C07281=1128.691,-66.097,-47.066,178.905,6.216,149.446
C07282=1128.696,-66.348,-47.056,178.902,6.216,149.447
C07283=1128.701,-66.597,-47.046,178.900,6.215,149.447
C07284=1128.707,-66.847,-47.035,178.898,6.215,149.448
C07285=1128.712,-67.097,-47.025,178.896,6.214,149.448
C07286=1128.717,-67.347,-47.015,178.893,6.213,149.449
C07287=1128.722,-67.596,-47.005,178.892,6.213,149.449
C07288=1128.727,-67.846,-46.994,178.890,6.212,149.450
C07289=1128.733,-68.096,-46.984,178.887,6.212,149.451
C07290=1128.739,-68.345,-46.974,178.885,6.211,149.451
C07291=1128.744,-68.595,-46.963,178.882,6.210,149.452
C07292=1128.749,-68.846,-46.954,178.880,6.210,149.452
C07293=1128.754,-69.095,-46.944,178.879,6.210,149.452
C07294=1128.760,-69.344,-46.934,178.877,6.209,149.453
C07295=1128.765,-69.595,-46.923,178.874,6.209,149.454
C07296=1128.770,-69.844,-46.913,178.872,6.208,149.454
C07297=1128.776,-70.094,-46.903,178.869,6.207,149.455
C07298=1128.781,-70.343,-46.893,178.867,6.206,149.455
C07299=1128.786,-70.593,-46.883,178.866,6.206,149.456
C07300=1128.792,-70.843,-46.873,178.863,6.206,149.456
C07301=1128.797,-71.093,-46.863,178.861,6.205,149.457
C07302=1128.802,-71.342,-46.854,178.859,6.204,149.457
C07303=1128.807,-71.592,-46.843,178.856,6.204,149.458
C07304=1128.813,-71.842,-46.833,178.855,6.204,149.458
C07305=1128.818,-72.091,-46.823,178.853,6.203,149.459
C07306=1128.824,-72.341,-46.814,178.850,6.202,149.459
C07307=1128.829,-72.591,-46.803,178.848,6.201,149.460
C07308=1128.834,-72.841,-46.793,178.846,6.201,149.460
C07309=1128.840,-73.091,-46.783,178.844,6.201,149.461
C07310=1128.845,-73.340,-46.773,178.842,6.200,149.461
C07311=1128.851,-73.590,-46.764,178.840,6.200,149.462
C07312=1128.856,-73.840,-46.753,178.837,6.199,149.462
C07313=1128.860,-74.089,-46.743,178.835,6.198,149.463
C07314=1128.866,-74.339,-46.733,178.834,6.198,149.463
C07315=1128.872,-74.589,-46.724,178.831,6.197,149.464
C07316=1128.877,-74.839,-46.713,178.829,6.197,149.464
C07317=1128.882,-75.089,-46.703,178.827,6.196,149.465
C07318=1128.887,-75.338,-46.693,178.824,6.195,149.465
C07319=1128.893,-75.588,-46.684,178.823,6.196,149.466
C07320=1128.898,-75.838,-46.674,178.821,6.195,149.466
C07321=1128.904,-76.087,-46.664,178.818,6.194,149.467
C07322=1128.909,-76.338,-46.654,178.816,6.193,149.467
C07323=1128.914,-76.587,-46.644,178.814,6.192,149.468
C07324=1128.920,-76.858,-46.633,178.812,6.193,149.469
C07325=1128.926,-77.130,-46.623,178.810,6.192,149.469
C07326=1128.931,-77.401,-46.612,178.808,6.191,149.470
C07327=1128.937,-77.674,-46.601,178.805,6.191,149.470
C07328=1128.943,-77.923,-46.591,178.803,6.190,149.471
C07329=1128.948,-78.173,-46.582,178.800,6.190,149.471
C07330=1128.954,-78.422,-46.572,178.798,6.189,149.472
C07331=1128.959,-78.672,-46.562,178.797,6.189,149.472
C07332=1128.965,-78.922,-46.553,178.794,6.188,149.473
C07333=1128.970,-79.171,-46.543,178.792,6.187,149.473
C07334=1128.975,-79.422,-46.533,178.790,6.187,149.474
C07335=1128.980,-79.672,-46.523,178.788,6.187,149.474
C07336=1128.985,-79.921,-46.514,178.786,6.186,149.475
C07337=1128.991,-80.171,-46.504,178.784,6.185,149.475
C07338=1128.997,-80.420,-46.494,178.781,6.185,149.476
C07339=1129.002,-80.670,-46.485,178.779,6.184,149.476
C07340=1129.007,-80.920,-46.475,178.778,6.184,149.477
C07341=1129.012,-81.169,-46.465,178.775,6.183,149.477
C07342=1129.018,-81.420,-46.455,178.773,6.183,149.478
C07343=1129.022,-81.669,-46.446,178.771,6.182,149.478
C07344=1129.028,-81.919,-46.436,178.769,6.182,149.479
C07345=1129.033,-82.169,-46.427,178.767,6.181,149.479
C07346=1129.039,-82.419,-46.417,178.765,6.181,149.480
C07347=1129.044,-82.668,-46.408,178.762,6.180,149.480
C07348=1129.050,-82.918,-46.398,178.761,6.180,149.481
C07349=1129.055,-83.168,-46.388,178.759,6.179,149.481
C07350=1129.061,-83.418,-46.379,178.756,6.178,149.482
C07351=1129.066,-83.667,-46.369,178.754,6.178,149.482
C07352=1129.071,-83.918,-46.359,178.753,6.178,149.483
C07353=1129.076,-84.167,-46.349,178.750,6.177,149.483
C07354=1129.082,-84.417,-46.340,178.748,6.176,149.484
C07355=1129.087,-84.667,-46.330,178.747,6.176,149.484
C07356=1129.092,-84.916,-46.321,178.744,6.176,149.485
C07357=1129.097,-85.166,-46.312,178.742,6.175,149.485
C07358=1129.103,-85.416,-46.302,178.740,6.174,149.486
C07359=1129.108,-85.665,-46.293,178.738,6.174,149.486
C07360=1129.114,-85.915,-46.283,178.736,6.174,149.487
C07361=1129.119,-86.165,-46.274,178.734,6.173,149.487
C07362=1129.125,-86.415,-46.264,178.731,6.172,149.488
C07363=1129.130,-86.664,-46.255,178.730,6.172,149.488
C07364=1129.135,-86.914,-46.245,178.728,6.171,149.489
C07365=1129.141,-87.164,-46.236,178.725,6.171,149.489
C07366=1129.146,-87.414,-46.227,178.723,6.170,149.490
C07367=1129.151,-87.663,-46.217,178.722,6.170,149.490
C07368=1129.156,-87.913,-46.208,178.719,6.170,149.491
C07369=1129.162,-88.163,-46.198,178.717,6.169,149.492
C07370=1129.167,-88.412,-46.189,178.715,6.169,149.492
C07371=1129.173,-88.663,-46.179,178.713,6.168,149.492
C07372=1129.178,-88.912,-46.170,178.711,6.167,149.493
C07373=1129.183,-89.162,-46.161,178.709,6.167,149.493
C07374=1129.189,-89.412,-46.151,178.707,6.167,149.494
C07375=1129.194,-89.661,-46.142,178.705,6.166,149.494
C07376=1129.199,-89.911,-46.133,178.703,6.165,149.495
C07377=1129.205,-90.161,-46.123,178.701,6.165,149.495
C07378=1129.210,-90.410,-46.114,178.699,6.165,149.496
C07379=1129.216,-90.661,-46.104,178.697,6.164,149.496
C07380=1129.221,-90.910,-46.095,178.695,6.164,149.497
C07381=1129.226,-91.160,-46.086,178.693,6.163,149.497
C07382=1129.232,-91.410,-46.076,178.690,6.163,149.498
C07383=1129.237,-91.660,-46.067,178.688,6.162,149.499
C07384=1129.242,-91.909,-46.058,178.686,6.162,149.499
C07385=1129.248,-92.159,-46.048,178.684,6.161,149.499
C07386=1129.253,-92.409,-46.039,178.682,6.161,149.500
C07387=1129.258,-92.659,-46.030,178.680,6.161,149.500
C07388=1129.264,-92.909,-46.021,178.678,6.160,149.501
C07389=1129.269,-93.158,-46.011,178.676,6.159,149.501
C07390=1129.274,-93.408,-46.002,178.674,6.159,149.502
C07391=1129.280,-93.658,-45.993,178.672,6.158,149.502
C07392=1129.285,-93.908,-45.984,178.670,6.158,149.503
C07393=1129.290,-94.157,-45.974,178.668,6.158,149.503
C07394=1129.296,-94.407,-45.965,178.666,6.157,149.504
C07395=1129.301,-94.657,-45.956,178.664,6.156,149.504
C07396=1129.306,-94.907,-45.947,178.662,6.155,149.505
C07397=1129.311,-95.157,-45.938,178.660,6.155,149.505
C07398=1129.317,-95.406,-45.928,178.658,6.155,149.506
C07399=1129.322,-95.656,-45.919,178.656,6.154,149.506
C07400=1129.328,-95.905,-45.911,178.654,6.154,149.507
C07401=1129.334,-96.156,-45.901,178.652,6.153,149.507
C07402=1129.339,-96.405,-45.892,178.649,6.153,149.508
C07403=1129.344,-96.655,-45.883,178.648,6.153,149.508
C07404=1129.349,-96.905,-45.874,178.646,6.152,149.509
C07405=1129.355,-97.155,-45.864,178.643,6.151,149.509
C07406=1129.360,-97.405,-45.855,178.642,6.151,149.510
C07407=1129.365,-97.654,-45.846,178.640,6.151,149.510
C07408=1129.370,-97.904,-45.837,178.637,6.150,149.511
C07409=1129.375,-98.154,-45.829,178.636,6.150,149.511
C07410=1129.382,-98.404,-45.819,178.634,6.149,149.512
C07411=1129.387,-98.653,-45.811,178.631,6.149,149.512
C07412=1129.392,-98.903,-45.802,178.630,6.149,149.513
C07413=1129.397,-99.153,-45.793,178.628,6.148,149.513
C07414=1129.403,-99.403,-45.783,178.625,6.147,149.514
C07415=1129.408,-99.653,-45.774,178.624,6.147,149.514
C07416=1129.413,-99.902,-45.765,178.622,6.146,149.515
C07417=1129.419,-100.152,-45.756,178.619,6.146,149.515
C07418=1129.424,-100.401,-45.747,178.618,6.146,149.516
C07419=1129.430,-100.652,-45.738,178.616,6.145,149.516
C07420=1129.435,-100.901,-45.729,178.614,6.145,149.517
C07421=1129.441,-101.151,-45.720,178.612,6.144,149.517
C07422=1129.446,-101.401,-45.711,178.610,6.143,149.518
C07423=1129.451,-101.651,-45.702,178.608,6.144,149.518
C07424=1129.457,-101.900,-45.694,178.606,6.143,149.519
C07425=1129.462,-102.150,-45.685,178.604,6.142,149.519
C07426=1129.468,-102.400,-45.675,178.602,6.142,149.520
C07427=1129.473,-102.650,-45.666,178.600,6.141,149.520
C07428=1129.479,-102.923,-45.657,178.598,6.141,149.521
C07429=1129.484,-103.195,-45.647,178.595,6.140,149.521
C07430=1129.490,-103.467,-45.637,178.593,6.140,149.522
C07431=1129.496,-103.739,-45.628,178.591,6.140,149.522
C07432=1129.502,-103.989,-45.619,178.589,6.139,149.523
C07433=1129.507,-104.239,-45.610,178.587,6.139,149.523
C07434=1129.512,-104.488,-45.601,178.585,6.138,149.524
C07435=1129.517,-104.738,-45.592,178.583,6.137,149.524
C07436=1129.523,-104.987,-45.584,178.581,6.137,149.525
C07437=1129.529,-105.238,-45.574,178.579,6.137,149.525
C07438=1129.534,-105.488,-45.566,178.577,6.136,149.526
C07439=1129.539,-105.738,-45.557,178.575,6.136,149.526
C07440=1129.545,-105.988,-45.548,178.573,6.135,149.527
C07441=1129.550,-106.237,-45.540,178.572,6.135,149.527
C07442=1129.555,-106.487,-45.531,178.569,6.135,149.528
C07443=1129.561,-106.737,-45.522,178.567,6.134,149.528
C07444=1129.566,-106.986,-45.513,178.566,6.134,149.529
C07445=1129.571,-107.236,-45.504,178.563,6.133,149.529
C07446=1129.577,-107.485,-45.496,178.561,6.132,149.530
C07447=1129.582,-107.736,-45.488,178.560,6.132,149.530
C07448=1129.587,-107.986,-45.479,178.557,6.132,149.531
C07449=1129.593,-108.236,-45.470,178.556,6.132,149.531
C07450=1129.598,-108.485,-45.461,178.554,6.131,149.532
C07451=1129.603,-108.735,-45.452,178.551,6.130,149.532
C07452=1129.609,-108.984,-45.443,178.550,6.130,149.533
C07453=1129.614,-109.235,-45.435,178.548,6.130,149.533
C07454=1129.620,-109.484,-45.427,178.546,6.130,149.533
C07455=1129.625,-109.734,-45.418,178.544,6.128,149.534
C07456=1129.630,-109.984,-45.409,178.542,6.128,149.534
C07457=1129.635,-110.234,-45.400,178.540,6.128,149.535
C07458=1129.641,-110.483,-45.392,178.538,6.127,149.535
C07459=1129.647,-110.733,-45.383,178.537,6.127,149.536
C07460=1129.652,-110.983,-45.374,178.535,6.126,149.536
C07461=1129.658,-111.232,-45.366,178.532,6.126,149.537
C07462=1129.663,-111.483,-45.358,178.531,6.126,149.537
C07463=1129.668,-111.733,-45.349,178.529,6.125,149.538
C07464=1129.673,-111.982,-45.340,178.527,6.125,149.538
C07465=1129.679,-112.232,-45.331,178.525,6.124,149.539
C07466=1129.685,-112.482,-45.323,178.523,6.123,149.539
C07467=1129.690,-112.732,-45.314,178.521,6.123,149.540
C07468=1129.696,-112.981,-45.306,178.519,6.123,149.540
C07469=1129.701,-113.231,-45.297,178.517,6.123,149.541
C07470=1129.706,-113.481,-45.289,178.515,6.122,149.541
C07471=1129.711,-113.731,-45.280,178.513,6.122,149.542
C07472=1129.717,-113.980,-45.271,178.511,6.121,149.542
C07473=1129.723,-114.231,-45.263,178.509,6.121,149.543
C07474=1129.728,-114.481,-45.254,178.507,6.121,149.543
C07475=1129.734,-114.730,-45.246,178.505,6.120,149.543
C07476=1129.738,-114.980,-45.238,178.504,6.120,149.544
C07477=1129.743,-115.230,-45.229,178.502,6.119,149.544
C07478=1129.749,-115.479,-45.221,178.500,6.118,149.545
C07479=1129.755,-115.729,-45.212,178.498,6.118,149.545
C07480=1129.760,-115.979,-45.204,178.496,6.117,149.546
C07481=1129.766,-116.228,-45.195,178.494,6.117,149.546
C07482=1129.771,-116.479,-45.187,178.492,6.117,149.547
C07483=1129.776,-116.729,-45.178,178.490,6.117,149.547
C07484=1129.782,-116.978,-45.169,178.488,6.116,149.548
C07485=1129.787,-117.228,-45.161,178.486,6.115,149.548
C07486=1129.792,-117.477,-45.153,178.484,6.115,149.549
C07487=1129.798,-117.728,-45.145,178.482,6.115,149.549
C07488=1129.803,-117.978,-45.136,178.481,6.115,149.550
C07489=1129.809,-118.227,-45.128,178.478,6.114,149.550
C07490=1129.814,-118.477,-45.119,178.477,6.114,149.551
C07491=1129.820,-118.727,-45.111,178.475,6.113,149.551
C07492=1129.826,-118.977,-45.103,178.474,6.113,149.551
C07493=1129.830,-119.226,-45.094,178.471,6.112,149.552
C07494=1129.836,-119.475,-45.086,178.469,6.111,149.552
C07495=1129.841,-119.726,-45.078,178.468,6.111,149.553
C07496=1129.846,-119.976,-45.069,178.465,6.111,149.553
C07497=1129.853,-120.226,-45.061,178.464,6.111,149.554
C07498=1129.857,-120.475,-45.053,178.462,6.110,149.554
C07499=1129.862,-120.726,-45.045,178.460,6.110,149.555
C07500=1129.868,-120.975,-45.036,178.458,6.109,149.555
C07501=1129.874,-121.225,-45.028,178.456,6.109,149.556
C07502=1129.879,-121.474,-45.019,178.454,6.109,149.556
C07503=1129.884,-121.725,-45.012,178.453,6.108,149.556
C07504=1129.889,-121.974,-45.003,178.451,6.107,149.557
C07505=1129.895,-122.224,-44.995,178.448,6.107,149.557
C07506=1129.901,-122.474,-44.986,178.447,6.107,149.558
C07507=1129.906,-122.723,-44.979,178.445,6.106,149.558
C07508=1129.911,-122.973,-44.970,178.443,6.106,149.559
C07509=1129.917,-123.223,-44.962,178.441,6.105,149.559
C07510=1129.922,-123.473,-44.953,178.439,6.105,149.560
C07511=1129.928,-123.723,-44.945,178.437,6.105,149.560
C07512=1129.933,-123.972,-44.937,178.436,6.104,149.561
C07513=1129.938,-124.223,-44.929,178.434,6.104,149.561
C07514=1129.944,-124.472,-44.921,178.432,6.104,149.562
C07515=1129.949,-124.722,-44.913,178.430,6.103,149.562
C07516=1129.955,-124.972,-44.905,178.428,6.103,149.563
C07517=1129.960,-125.222,-44.896,178.426,6.102,149.563
C07518=1129.966,-125.471,-44.888,178.425,6.102,149.564
C07519=1129.971,-125.721,-44.880,178.422,6.102,149.564
C07520=1129.976,-125.971,-44.872,178.420,6.101,149.565
C07521=1129.982,-126.221,-44.864,178.419,6.100,149.565
C07522=1129.986,-126.471,-44.856,178.417,6.100,149.565
C07523=1129.993,-126.720,-44.848,178.415,6.100,149.566
C07524=1129.998,-126.970,-44.839,178.413,6.099,149.566
C07525=1130.004,-127.220,-44.831,178.411,6.099,149.567
C07526=1130.009,-127.470,-44.824,178.409,6.098,149.567
C07527=1130.014,-127.719,-44.815,178.408,6.098,149.568
C07528=1130.020,-127.970,-44.807,178.405,6.098,149.568
C07529=1130.025,-128.219,-44.800,178.404,6.097,149.568
C07530=1130.030,-128.469,-44.791,178.402,6.097,149.569
C07531=1130.036,-128.719,-44.783,178.401,6.097,149.569
C07532=1129.615,-128.730,-44.827,178.397,6.100,149.571
C07533=1129.610,-128.481,-44.836,178.399,6.101,149.571
C07534=1129.604,-128.230,-44.844,178.401,6.101,149.570
C07535=1129.599,-127.981,-44.851,178.403,6.101,149.570
C07536=1129.594,-127.731,-44.860,178.404,6.101,149.569
C07537=1129.587,-127.481,-44.868,178.407,6.102,149.569
C07538=1129.583,-127.231,-44.875,178.408,6.102,149.569
C07539=1129.577,-126.982,-44.884,178.410,6.103,149.568
C07540=1129.571,-126.732,-44.892,178.411,6.103,149.568
C07541=1129.567,-126.482,-44.900,178.414,6.104,149.567
C07542=1129.561,-126.232,-44.908,178.416,6.105,149.567
C07543=1129.556,-125.982,-44.916,178.417,6.104,149.566
C07544=1129.550,-125.733,-44.925,178.420,6.105,149.566
C07545=1129.545,-125.483,-44.932,178.421,6.105,149.565
C07546=1129.539,-125.233,-44.941,178.423,6.106,149.565
C07547=1129.534,-124.983,-44.949,178.425,6.106,149.564
C07548=1129.528,-124.733,-44.956,178.427,6.107,149.564
C07549=1129.523,-124.484,-44.965,178.428,6.107,149.563
C07550=1129.517,-124.234,-44.973,178.431,6.108,149.563
C07551=1129.512,-123.984,-44.982,178.432,6.108,149.562
C07552=1129.507,-123.734,-44.990,178.434,6.108,149.562
C07553=1129.502,-123.485,-44.998,178.436,6.108,149.561
C07554=1129.496,-123.234,-45.006,178.438,6.109,149.561
C07555=1129.490,-122.985,-45.015,178.439,6.109,149.561
C07556=1129.486,-122.735,-45.022,178.441,6.110,149.560
C07557=1129.479,-122.485,-45.030,178.443,6.110,149.560
C07558=1129.474,-122.235,-45.039,178.445,6.111,149.559
C07559=1129.469,-121.985,-45.047,178.447,6.112,149.559
C07560=1129.463,-121.736,-45.056,178.449,6.112,149.558
C07561=1129.458,-121.485,-45.063,178.451,6.112,149.558
C07562=1129.453,-121.236,-45.072,178.453,6.112,149.557
C07563=1129.447,-120.986,-45.081,178.455,6.113,149.557
C07564=1129.442,-120.736,-45.089,178.456,6.113,149.557
C07565=1129.437,-120.487,-45.097,178.458,6.114,149.556
C07566=1129.431,-120.237,-45.105,178.460,6.114,149.556
C07567=1129.426,-119.988,-45.114,178.462,6.115,149.555
C07568=1129.420,-119.737,-45.122,178.464,6.115,149.555
C07569=1129.415,-119.487,-45.131,178.466,6.115,149.554
C07570=1129.409,-119.237,-45.139,178.468,6.116,149.554
C07571=1129.405,-118.988,-45.147,178.470,6.116,149.553
C07572=1129.398,-118.738,-45.155,178.472,6.117,149.553
C07573=1129.393,-118.488,-45.164,178.474,6.117,149.552
C07574=1129.388,-118.238,-45.173,178.476,6.118,149.552
C07575=1129.382,-117.989,-45.180,178.477,6.118,149.551
C07576=1129.377,-117.739,-45.189,178.479,6.119,149.551
C07577=1129.372,-117.489,-45.197,178.481,6.119,149.550
C07578=1129.366,-117.240,-45.205,178.483,6.119,149.550
C07579=1129.361,-116.990,-45.214,178.485,6.120,149.549
C07580=1129.356,-116.739,-45.222,178.487,6.120,149.549
C07581=1129.350,-116.490,-45.231,178.489,6.121,149.548
C07582=1129.345,-116.240,-45.239,178.490,6.121,149.548
C07583=1129.339,-115.990,-45.248,178.493,6.121,149.548
C07584=1129.334,-115.741,-45.257,178.495,6.122,149.547
C07585=1129.328,-115.490,-45.265,178.496,6.122,149.547
C07586=1129.323,-115.241,-45.273,178.499,6.123,149.546
C07587=1129.318,-114.991,-45.282,178.500,6.123,149.546
C07588=1129.312,-114.741,-45.290,178.502,6.124,149.545
C07589=1129.307,-114.492,-45.298,178.504,6.124,149.545
C07590=1129.301,-114.242,-45.307,178.506,6.125,149.544
C07591=1129.296,-113.991,-45.315,178.508,6.125,149.544
C07592=1129.291,-113.742,-45.324,178.510,6.125,149.543
C07593=1129.285,-113.492,-45.333,178.512,6.126,149.543
C07594=1129.280,-113.243,-45.342,178.513,6.126,149.542
C07595=1129.274,-112.992,-45.350,178.516,6.127,149.542
C07596=1129.269,-112.743,-45.358,178.517,6.127,149.541
C07597=1129.264,-112.493,-45.367,178.519,6.127,149.541
C07598=1129.258,-112.243,-45.376,178.522,6.128,149.540
C07599=1129.252,-111.994,-45.384,178.523,6.128,149.540
C07600=1129.247,-111.744,-45.393,178.525,6.129,149.539
C07601=1129.242,-111.494,-45.402,178.527,6.129,149.539
C07602=1129.236,-111.243,-45.410,178.529,6.130,149.538
C07603=1129.231,-110.995,-45.418,178.531,6.130,149.538
C07604=1129.226,-110.745,-45.427,178.533,6.130,149.538
C07605=1129.221,-110.495,-45.436,178.535,6.131,149.537
C07606=1129.215,-110.245,-45.444,178.537,6.131,149.537
C07607=1129.210,-109.995,-45.452,178.539,6.132,149.536
C07608=1129.205,-109.745,-45.461,178.541,6.132,149.536
C07609=1129.200,-109.495,-45.470,178.543,6.132,149.535
C07610=1129.194,-109.246,-45.479,178.545,6.133,149.535
C07611=1129.189,-108.997,-45.488,178.546,6.134,149.534
C07612=1129.183,-108.746,-45.496,178.548,6.134,149.534
C07613=1129.178,-108.496,-45.505,178.550,6.135,149.533
C07614=1129.171,-108.247,-45.514,178.552,6.135,149.533
C07615=1129.166,-107.997,-45.523,178.554,6.136,149.532
C07616=1129.161,-107.747,-45.532,178.556,6.136,149.532
C07617=1129.156,-107.497,-45.541,178.558,6.136,149.531
C07618=1129.150,-107.247,-45.548,178.560,6.137,149.531
C07619=1129.145,-106.998,-45.557,178.562,6.137,149.530
C07620=1129.140,-106.748,-45.566,178.564,6.138,149.530
C07621=1129.134,-106.498,-45.575,178.566,6.139,149.529
C07622=1129.129,-106.248,-45.584,178.568,6.139,149.529
C07623=1129.123,-105.999,-45.593,178.570,6.139,149.528
C07624=1129.118,-105.749,-45.601,178.572,6.139,149.528
C07625=1129.113,-105.499,-45.610,178.574,6.140,149.528
C07626=1129.108,-105.249,-45.619,178.576,6.141,149.527
C07627=1129.102,-105.000,-45.627,178.578,6.141,149.527
C07628=1129.097,-104.750,-45.636,178.580,6.141,149.526
C07629=1129.092,-104.500,-45.645,178.582,6.142,149.526
C07630=1129.086,-104.250,-45.654,178.584,6.142,149.525
C07631=1129.080,-104.000,-45.663,178.586,6.143,149.525
C07632=1129.075,-103.750,-45.672,178.587,6.143,149.524
C07633=1129.069,-103.478,-45.681,178.590,6.144,149.524
C07634=1129.063,-103.206,-45.692,178.592,6.144,149.523
C07635=1129.058,-102.934,-45.701,178.594,6.145,149.522
C07636=1129.052,-102.661,-45.711,178.597,6.145,149.522
C07637=1129.047,-102.411,-45.719,178.598,6.145,149.521
C07638=1129.041,-102.161,-45.728,178.600,6.146,149.521
C07639=1129.036,-101.912,-45.737,178.603,6.147,149.520
C07640=1129.030,-101.662,-45.746,178.604,6.147,149.520
C07641=1129.025,-101.412,-45.755,178.606,6.148,149.519
C07642=1129.019,-101.162,-45.764,178.608,6.147,149.519
C07643=1129.014,-100.913,-45.773,178.610,6.148,149.519
C07644=1129.009,-100.663,-45.782,178.612,6.149,149.518
C07645=1129.004,-100.413,-45.791,178.614,6.149,149.518
C07646=1128.997,-100.163,-45.800,178.616,6.150,149.517
C07647=1128.992,-99.913,-45.809,178.618,6.150,149.517
C07648=1128.987,-99.664,-45.818,178.620,6.150,149.516
C07649=1128.982,-99.414,-45.827,178.622,6.151,149.516
C07650=1128.977,-99.165,-45.836,178.624,6.152,149.515
C07651=1128.971,-98.914,-45.846,178.626,6.152,149.515
C07652=1128.966,-98.665,-45.855,178.628,6.153,149.514
C07653=1128.961,-98.415,-45.864,178.630,6.153,149.514
C07654=1128.955,-98.166,-45.872,178.632,6.153,149.513
C07655=1128.950,-97.916,-45.881,178.634,6.154,149.513
C07656=1128.944,-97.666,-45.890,178.636,6.155,149.512
C07657=1128.939,-97.416,-45.899,178.638,6.155,149.512
C07658=1128.934,-97.166,-45.908,178.640,6.155,149.511
C07659=1128.929,-96.916,-45.917,178.642,6.156,149.511
C07660=1128.923,-96.666,-45.927,178.644,6.156,149.510
C07661=1128.918,-96.417,-45.936,178.646,6.157,149.510
C07662=1128.913,-96.167,-45.945,178.648,6.158,149.509
C07663=1128.907,-95.918,-45.954,178.650,6.158,149.509
C07664=1128.901,-95.667,-45.963,178.652,6.158,149.508
C07665=1128.896,-95.418,-45.972,178.654,6.159,149.508
C07666=1128.891,-95.168,-45.982,178.656,6.159,149.507
C07667=1128.886,-94.918,-45.991,178.659,6.159,149.507
C07668=1128.880,-94.668,-46.000,178.661,6.160,149.506
C07669=1128.875,-94.418,-46.009,178.662,6.160,149.506
C07670=1128.870,-94.169,-46.018,178.665,6.161,149.505
C07671=1128.864,-93.918,-46.027,178.667,6.162,149.505
C07672=1128.859,-93.669,-46.037,178.669,6.162,149.504
C07673=1128.854,-93.419,-46.046,178.671,6.162,149.504
C07674=1128.848,-93.169,-46.055,178.673,6.163,149.503
C07675=1128.843,-92.919,-46.064,178.675,6.164,149.503
C07676=1128.838,-92.670,-46.074,178.677,6.164,149.502
C07677=1128.832,-92.420,-46.083,178.679,6.165,149.502
C07678=1128.827,-92.170,-46.092,178.681,6.165,149.501
C07679=1128.821,-91.921,-46.101,178.683,6.165,149.501
C07680=1128.815,-91.671,-46.111,178.685,6.166,149.500
C07681=1128.810,-91.422,-46.120,178.687,6.167,149.500
C07682=1128.805,-91.172,-46.129,178.688,6.167,149.499
C07683=1128.799,-90.922,-46.138,178.691,6.167,149.499
C07684=1128.794,-90.672,-46.148,178.693,6.168,149.498
C07685=1128.789,-90.422,-46.157,178.695,6.169,149.498
C07686=1128.783,-90.172,-46.166,178.697,6.169,149.497
C07687=1128.778,-89.923,-46.176,178.699,6.169,149.497
C07688=1128.773,-89.673,-46.185,178.702,6.170,149.496
C07689=1128.767,-89.423,-46.194,178.703,6.170,149.496
C07690=1128.762,-89.174,-46.204,178.705,6.171,149.495
C07691=1128.756,-88.924,-46.213,178.708,6.171,149.495
C07692=1128.751,-88.674,-46.222,178.710,6.172,149.494
C07693=1128.746,-88.425,-46.232,178.711,6.172,149.494
C07694=1128.740,-88.174,-46.241,178.714,6.173,149.493
C07695=1128.736,-87.925,-46.251,178.716,6.174,149.493
C07696=1128.730,-87.675,-46.261,178.717,6.174,149.492
C07697=1128.724,-87.425,-46.269,178.720,6.174,149.492
C07698=1128.719,-87.175,-46.280,178.722,6.175,149.491
C07699=1128.714,-86.925,-46.289,178.724,6.176,149.491
C07700=1128.709,-86.675,-46.298,178.725,6.176,149.490
C07701=1128.704,-86.426,-46.308,178.728,6.176,149.490
C07702=1128.698,-86.176,-46.317,178.730,6.177,149.489
C07703=1128.693,-85.926,-46.327,178.733,6.178,149.489
C07704=1128.688,-85.676,-46.336,178.734,6.178,149.488
C07705=1128.682,-85.427,-46.346,178.736,6.178,149.488
C07706=1128.677,-85.177,-46.355,178.739,6.179,149.487
C07707=1128.671,-84.927,-46.365,178.740,6.179,149.487
C07708=1128.666,-84.678,-46.374,178.742,6.180,149.486
C07709=1128.661,-84.428,-46.383,178.745,6.181,149.486
C07710=1128.655,-84.178,-46.393,178.747,6.181,149.485
C07711=1128.650,-83.928,-46.402,178.748,6.181,149.485
C07712=1128.645,-83.679,-46.412,178.751,6.182,149.484
C07713=1128.639,-83.429,-46.421,178.753,6.182,149.484
C07714=1128.634,-83.179,-46.432,178.755,6.183,149.483
C07715=1128.629,-82.929,-46.441,178.757,6.183,149.483
C07716=1128.624,-82.679,-46.451,178.759,6.184,149.482
C07717=1128.618,-82.429,-46.461,178.761,6.185,149.482
C07718=1128.613,-82.180,-46.470,178.764,6.185,149.481
C07719=1128.607,-81.930,-46.480,178.765,6.185,149.481
C07720=1128.602,-81.681,-46.489,178.767,6.186,149.480
C07721=1128.597,-81.431,-46.499,178.770,6.187,149.480
C07722=1128.591,-81.181,-46.508,178.772,6.188,149.479
C07723=1128.586,-80.932,-46.519,178.774,6.187,149.479
C07724=1128.581,-80.681,-46.528,178.776,6.188,149.478
C07725=1128.576,-80.432,-46.538,178.778,6.189,149.478
C07726=1128.570,-80.182,-46.547,178.780,6.190,149.477
C07727=1128.565,-79.932,-46.557,178.782,6.189,149.477
C07728=1128.559,-79.683,-46.567,178.784,6.190,149.476
C07729=1128.554,-79.433,-46.576,178.786,6.191,149.476
C07730=1128.548,-79.183,-46.586,178.789,6.192,149.475
C07731=1128.543,-78.933,-46.595,178.791,6.192,149.475
C07732=1128.538,-78.683,-46.606,178.793,6.192,149.474
C07733=1128.533,-78.434,-46.616,178.795,6.193,149.474
C07734=1128.528,-78.184,-46.625,178.797,6.194,149.473
C07735=1128.522,-77.934,-46.635,178.799,6.194,149.473
C07736=1128.516,-77.685,-46.645,178.801,6.194,149.472
C07737=1128.511,-77.413,-46.656,178.803,6.195,149.472
C07738=1128.505,-77.141,-46.666,178.806,6.195,149.471
C07739=1128.499,-76.870,-46.677,178.808,6.196,149.470
C07740=1128.493,-76.598,-46.687,178.810,6.197,149.470
C07741=1128.488,-76.348,-46.698,178.812,6.198,149.469
C07742=1128.483,-76.099,-46.707,178.815,6.198,149.469
C07743=1128.477,-75.849,-46.717,178.817,6.199,149.468
C07744=1128.472,-75.599,-46.727,178.819,6.199,149.468
C07745=1128.467,-75.350,-46.737,178.821,6.200,149.467
C07746=1128.462,-75.100,-46.747,178.823,6.200,149.467
C07747=1128.456,-74.850,-46.757,178.826,6.201,149.466
C07748=1128.450,-74.600,-46.767,178.827,6.201,149.466
C07749=1128.446,-74.350,-46.777,178.829,6.202,149.465
C07750=1128.440,-74.101,-46.787,178.832,6.202,149.465
C07751=1128.434,-73.851,-46.796,178.834,6.203,149.464
C07752=1128.429,-73.601,-46.806,178.836,6.204,149.464
C07753=1128.424,-73.352,-46.816,178.838,6.204,149.463
C07754=1128.419,-73.102,-46.827,178.840,6.204,149.463
C07755=1128.413,-72.851,-46.836,178.842,6.205,149.462
C07756=1128.408,-72.602,-46.846,178.845,6.206,149.462
C07757=1128.402,-72.353,-46.856,178.847,6.207,149.461
C07758=1128.397,-72.102,-46.867,178.849,6.207,149.461
C07759=1128.392,-71.853,-46.877,178.851,6.207,149.460
C07760=1128.387,-71.603,-46.886,178.853,6.208,149.460
C07761=1128.381,-71.354,-46.896,178.855,6.208,149.459
C07762=1128.376,-71.103,-46.907,178.858,6.209,149.459
C07763=1128.370,-70.854,-46.917,178.860,6.210,149.458
C07764=1128.366,-70.605,-46.926,178.861,6.210,149.458
C07765=1128.360,-70.355,-46.937,178.864,6.211,149.457
C07766=1128.355,-70.105,-46.947,178.866,6.211,149.456
C07767=1128.349,-69.855,-46.957,178.868,6.212,149.456
C07768=1128.344,-69.605,-46.966,178.871,6.213,149.455
C07769=1128.339,-69.356,-46.977,178.873,6.213,149.455
C07770=1128.334,-69.106,-46.987,178.874,6.213,149.455
C07771=1128.328,-68.856,-46.997,178.877,6.214,149.454
C07772=1128.322,-68.606,-47.007,178.879,6.215,149.454
C07773=1128.318,-68.357,-47.017,178.881,6.215,149.453
C07774=1128.313,-68.107,-47.028,178.884,6.216,149.452
C07775=1128.307,-67.857,-47.038,178.885,6.216,149.452
C07776=1128.301,-67.608,-47.048,178.887,6.217,149.451
C07777=1128.296,-67.358,-47.059,178.890,6.217,149.451
C07778=1128.291,-67.108,-47.069,178.892,6.218,149.450
C07779=1128.286,-66.859,-47.079,178.894,6.219,149.450
C07780=1128.281,-66.608,-47.088,178.897,6.219,149.449
C07781=1128.275,-66.358,-47.099,178.899,6.220,149.449
C07782=1128.269,-66.109,-47.109,178.900,6.220,149.448
C07783=1128.264,-65.859,-47.119,178.903,6.221,149.448
C07784=1128.259,-65.609,-47.130,178.905,6.222,149.447
C07785=1128.253,-65.360,-47.140,178.907,6.222,149.447
C07786=1128.249,-65.110,-47.150,178.910,6.223,149.446
C07787=1128.243,-64.860,-47.160,178.912,6.223,149.446
C07788=1128.238,-64.611,-47.171,178.914,6.223,149.445
C07789=1128.233,-64.361,-47.181,178.916,6.224,149.445
C07790=1128.227,-64.111,-47.192,178.918,6.225,149.444
C07791=1128.222,-63.862,-47.202,178.920,6.226,149.444
C07792=1128.217,-63.612,-47.212,178.923,6.226,149.443
C07793=1128.211,-63.362,-47.223,178.925,6.227,149.443
C07794=1128.206,-63.113,-47.233,178.927,6.228,149.442
C07795=1128.201,-62.862,-47.243,178.929,6.228,149.442
C07796=1128.195,-62.613,-47.254,178.931,6.228,149.441
C07797=1128.190,-62.364,-47.263,178.933,6.229,149.441
C07798=1128.185,-62.113,-47.274,178.936,6.229,149.440
C07799=1128.180,-61.864,-47.284,178.938,6.230,149.439
C07800=1128.175,-61.613,-47.295,178.940,6.231,149.439
C07801=1128.169,-61.365,-47.306,178.942,6.232,149.438
C07802=1128.164,-61.115,-47.316,178.945,6.233,149.438
C07803=1128.159,-60.865,-47.326,178.946,6.232,149.438
C07804=1128.153,-60.615,-47.337,178.949,6.233,149.437
C07805=1128.148,-60.365,-47.347,178.951,6.234,149.436
C07806=1128.143,-60.115,-47.357,178.953,6.234,149.436
C07807=1128.137,-59.866,-47.368,178.955,6.235,149.435
C07808=1128.132,-59.616,-47.379,178.958,6.236,149.435
C07809=1128.127,-59.367,-47.389,178.960,6.236,149.434
C07810=1128.122,-59.116,-47.400,178.962,6.237,149.434
C07811=1128.116,-58.867,-47.410,178.965,6.238,149.433
C07812=1128.111,-58.617,-47.420,178.966,6.238,149.433
C07813=1128.106,-58.368,-47.431,178.968,6.239,149.432
C07814=1128.100,-58.118,-47.442,178.971,6.239,149.432
C07815=1128.095,-57.868,-47.452,178.973,6.240,149.431
C07816=1128.090,-57.618,-47.462,178.976,6.240,149.431
C07817=1128.085,-57.369,-47.474,178.978,6.241,149.430
C07818=1128.079,-57.119,-47.484,178.980,6.242,149.430
C07819=1128.074,-56.869,-47.494,178.982,6.243,149.429
C07820=1128.069,-56.619,-47.505,178.985,6.243,149.428
C07821=1128.061,-56.267,-47.520,178.987,6.243,149.428
C07822=1128.034,-54.962,-47.575,179.507,5.297,149.069
C07823=1128.029,-54.712,-47.586,179.507,5.301,149.069
C07824=1128.024,-54.462,-47.596,179.507,5.306,149.071
C07825=1128.018,-54.213,-47.606,179.506,5.311,149.072
C07826=1128.013,-53.964,-47.617,179.507,5.315,149.073
C07827=1128.008,-53.713,-47.628,179.506,5.321,149.074
C07828=1128.002,-53.464,-47.638,179.506,5.325,149.075
C07829=1127.997,-53.214,-47.649,179.506,5.330,149.076
C07830=1127.991,-52.964,-47.659,179.505,5.334,149.077
C07831=1127.986,-52.714,-47.671,179.505,5.339,149.078
C07832=1127.980,-52.465,-47.681,179.505,5.344,149.079
C07833=1127.975,-52.215,-47.691,179.505,5.348,149.080
C07834=1127.970,-51.966,-47.702,179.504,5.353,149.081
C07835=1127.965,-51.716,-47.713,179.504,5.358,149.083
C07836=1127.960,-51.466,-47.723,179.505,5.363,149.083
C07837=1127.954,-51.216,-47.733,179.504,5.367,149.085
C07838=1127.949,-50.967,-47.745,179.504,5.372,149.086
C07839=1127.944,-50.717,-47.755,179.503,5.376,149.087
C07840=1127.939,-50.467,-47.766,179.504,5.381,149.088
C07841=1127.933,-50.218,-47.776,179.503,5.385,149.089
C07842=1127.928,-49.968,-47.787,179.503,5.391,149.090
C07843=1127.922,-49.718,-47.798,179.503,5.395,149.091
C07844=1127.917,-49.468,-47.809,179.503,5.400,149.092
C07845=1127.912,-49.219,-47.819,179.503,5.405,149.093
C07846=1127.907,-48.968,-47.830,179.502,5.409,149.094
C07847=1127.901,-48.719,-47.841,179.502,5.414,149.095
C07848=1127.896,-48.469,-47.851,179.502,5.418,149.096
C07849=1127.891,-48.220,-47.862,179.502,5.423,149.098
C07850=1127.882,-47.814,-47.880,179.502,5.431,149.099
C07851=1127.874,-47.408,-47.897,179.501,5.439,149.101
C07852=1127.865,-47.003,-47.915,179.500,5.446,149.103
C07853=1127.856,-46.597,-47.932,179.501,5.454,149.104
C07854=1127.851,-46.348,-47.943,179.501,5.459,149.106
C07855=1127.846,-46.098,-47.954,179.500,5.463,149.107
C07856=1127.840,-45.848,-47.964,179.500,5.468,149.108
C07857=1127.836,-45.599,-47.975,179.500,5.473,149.109
C07858=1127.829,-45.349,-47.986,179.500,5.477,149.110
C07859=1127.825,-45.099,-47.998,179.500,5.482,149.111
C07860=1127.820,-44.849,-48.008,179.499,5.486,149.112
C07861=1127.814,-44.600,-48.019,179.499,5.492,149.113
C07862=1127.809,-44.350,-48.030,179.499,5.496,149.114
C07863=1127.803,-44.101,-48.041,179.499,5.501,149.115
C07864=1127.798,-43.850,-48.052,179.499,5.506,149.116
C07865=1127.793,-43.602,-48.063,179.498,5.510,149.117
C07866=1127.787,-43.351,-48.074,179.498,5.515,149.119
C07867=1127.783,-43.101,-48.085,179.499,5.520,149.119
C07868=1127.777,-42.852,-48.095,179.501,5.526,149.120
C07869=1127.772,-42.602,-48.107,179.503,5.532,149.121
C07870=1127.766,-42.353,-48.118,179.505,5.538,149.121
C07871=1127.761,-42.103,-48.129,179.507,5.544,149.122
C07872=1127.757,-41.853,-48.140,179.508,5.549,149.123
C07873=1127.750,-41.603,-48.151,179.510,5.555,149.124
C07874=1127.746,-41.354,-48.162,179.513,5.561,149.124
C07875=1127.741,-41.104,-48.173,179.514,5.566,149.125
C07876=1127.735,-40.854,-48.184,179.516,5.572,149.126
C07877=1127.730,-40.605,-48.195,179.518,5.578,149.126
C07878=1127.725,-40.356,-48.206,179.519,5.583,149.127
C07879=1127.719,-40.105,-48.218,179.521,5.589,149.128
C07880=1127.714,-39.855,-48.229,179.522,5.594,149.129
C07881=1127.709,-39.605,-48.241,179.524,5.599,149.129
C07882=1127.703,-39.357,-48.252,179.526,5.605,149.130
C07883=1127.698,-39.106,-48.262,179.527,5.610,149.131
C07884=1127.693,-38.856,-48.274,179.528,5.615,149.131
C07885=1127.688,-38.607,-48.285,179.530,5.620,149.132
C07886=1127.682,-38.358,-48.297,179.531,5.626,149.133
C07887=1127.678,-38.108,-48.308,179.532,5.631,149.134
C07888=1127.671,-37.858,-48.319,179.534,5.636,149.134
C07889=1127.667,-37.608,-48.330,179.535,5.641,149.135
C07890=1127.661,-37.358,-48.342,179.536,5.646,149.136
C07891=1127.656,-37.109,-48.354,179.537,5.651,149.137
C07892=1127.650,-36.860,-48.365,179.538,5.656,149.137
C07893=1127.646,-36.610,-48.376,179.539,5.660,149.138
C07894=1127.640,-36.360,-48.388,179.540,5.666,149.139
C07895=1127.636,-36.110,-48.399,179.541,5.670,149.140
C07896=1127.629,-35.861,-48.410,179.542,5.675,149.140
C07897=1127.625,-35.611,-48.422,179.543,5.680,149.141
C07898=1127.619,-35.361,-48.433,179.543,5.685,149.142
C07899=1127.614,-35.111,-48.445,179.544,5.689,149.143
C07900=1127.609,-34.861,-48.457,179.545,5.694,149.144
C07901=1127.604,-34.613,-48.468,179.545,5.699,149.145
C07902=1127.599,-34.397,-48.479,179.545,5.702,149.145
C07903=1127.595,-34.181,-48.488,179.546,5.707,149.146
C07904=1127.591,-33.966,-48.498,179.547,5.710,149.147
C07905=1127.585,-33.750,-48.508,179.546,5.714,149.147
C07906=1127.581,-33.535,-48.518,179.547,5.719,149.148
C07907=1127.576,-33.318,-48.528,179.548,5.722,149.149
C07908=1127.572,-33.103,-48.538,179.548,5.726,149.150
C07909=1127.567,-32.888,-48.548,179.548,5.730,149.150
C07910=1127.562,-32.638,-48.560,179.548,5.734,149.151
C07911=1127.557,-32.388,-48.571,179.548,5.738,149.152
C07912=1127.552,-32.138,-48.583,179.549,5.743,149.153
C07913=1127.546,-31.889,-48.595,179.549,5.747,149.154
C07914=1127.542,-31.640,-48.607,179.548,5.751,149.155
C07915=1127.537,-31.390,-48.618,179.549,5.756,149.156
C07916=1127.531,-31.140,-48.630,179.549,5.760,149.157
C07917=1127.526,-30.891,-48.641,179.548,5.764,149.158
C07918=1127.520,-30.641,-48.653,179.548,5.768,149.159
C07919=1127.515,-30.391,-48.665,179.548,5.772,149.160
C07920=1127.510,-30.141,-48.676,179.547,5.776,149.161
C07921=1127.505,-29.891,-48.688,179.547,5.780,149.162
C07922=1127.499,-29.641,-48.700,179.546,5.785,149.163
C07923=1127.494,-29.393,-48.712,179.546,5.789,149.164
C07924=1127.489,-29.143,-48.724,179.546,5.793,149.165
C07925=1127.484,-28.893,-48.736,179.546,5.797,149.166
C07926=1127.479,-28.644,-48.747,179.545,5.801,149.167
C07927=1127.473,-28.394,-48.759,179.544,5.805,149.168
C07928=1127.468,-28.144,-48.771,179.543,5.809,149.169
C07929=1127.463,-27.894,-48.782,179.542,5.812,149.170
C07930=1127.458,-27.645,-48.794,179.542,5.817,149.171
C07931=1127.453,-27.395,-48.806,179.541,5.821,149.172
C07932=1127.447,-27.146,-48.818,179.540,5.824,149.173
C07933=1127.442,-26.896,-48.829,179.539,5.828,149.175
C07934=1127.437,-26.646,-48.841,179.538,5.832,149.176
C07935=1127.431,-26.396,-48.853,179.536,5.836,149.177
C07936=1127.427,-26.147,-48.865,179.535,5.840,149.178
C07937=1127.421,-25.897,-48.877,179.536,5.844,149.179
C07938=1127.416,-25.647,-48.889,179.536,5.849,149.180
C07939=1127.411,-25.397,-48.901,179.537,5.855,149.181
C07940=1127.406,-25.148,-48.912,179.538,5.859,149.182
C07941=1127.401,-24.898,-48.924,179.538,5.864,149.183
C07942=1127.395,-24.648,-48.936,179.540,5.869,149.183
C07943=1127.390,-24.398,-48.948,179.540,5.874,149.184
C07944=1127.385,-24.150,-48.959,179.541,5.880,149.185
C07945=1127.379,-23.900,-48.972,179.542,5.884,149.186
C07946=1127.374,-23.650,-48.984,179.542,5.889,149.187
C07947=1127.369,-23.400,-48.996,179.544,5.894,149.188
C07948=1127.363,-23.151,-49.008,179.544,5.899,149.188
C07949=1127.359,-22.901,-49.019,179.545,5.904,149.189
C07950=1127.353,-22.651,-49.031,179.546,5.909,149.190
C07951=1127.348,-22.402,-49.044,179.547,5.914,149.191
C07952=1127.343,-22.152,-49.056,179.547,5.918,149.192
C07953=1127.337,-21.902,-49.068,179.548,5.924,149.193
C07954=1127.332,-21.653,-49.080,179.549,5.929,149.194
C07955=1127.328,-21.403,-49.092,179.550,5.933,149.194
C07956=1127.322,-21.153,-49.103,179.550,5.938,149.195
C07957=1127.317,-20.904,-49.116,179.551,5.943,149.196
C07958=1127.313,-20.688,-49.127,179.552,5.947,149.197
C07959=1127.308,-20.473,-49.137,179.553,5.951,149.197
C07960=1127.304,-20.257,-49.148,179.554,5.956,149.198
C07961=1127.298,-20.042,-49.158,179.553,5.959,149.199
C07962=1127.295,-19.826,-49.168,179.554,5.964,149.200
C07963=1127.289,-19.611,-49.179,179.555,5.968,149.200
C07964=1127.286,-19.395,-49.189,179.556,5.972,149.201
C07965=1127.281,-19.180,-49.200,179.557,5.976,149.202
C07966=1127.276,-18.931,-49.212,179.557,5.981,149.202
C07967=1127.270,-18.681,-49.224,179.558,5.986,149.203
C07968=1127.265,-18.432,-49.237,179.559,5.991,149.204
C07969=1127.260,-18.182,-49.249,179.560,5.995,149.205
C07970=1127.254,-17.932,-49.261,179.560,6.000,149.206
C07971=1127.250,-17.682,-49.274,179.561,6.005,149.207
C07972=1127.244,-17.432,-49.286,179.562,6.009,149.207
C07973=1127.239,-17.182,-49.298,179.563,6.015,149.208
C07974=1127.234,-16.933,-49.311,179.563,6.020,149.209
C07975=1127.229,-16.684,-49.323,179.564,6.024,149.210
C07976=1127.223,-16.434,-49.335,179.565,6.029,149.211
C07977=1127.218,-16.185,-49.348,179.565,6.033,149.212
C07978=1127.213,-15.935,-49.360,179.566,6.038,149.212
C07979=1127.208,-15.685,-49.372,179.567,6.043,149.213
C07980=1127.203,-15.436,-49.385,179.568,6.048,149.214
C07981=1127.198,-15.185,-49.397,179.569,6.052,149.215
C07982=1127.193,-14.936,-49.410,179.569,6.057,149.216
C07983=1127.188,-14.687,-49.422,179.570,6.062,149.216
C07984=1127.182,-14.437,-49.434,179.571,6.066,149.217
C07985=1127.177,-14.187,-49.447,179.571,6.071,149.218
C07986=1127.172,-13.938,-49.459,179.572,6.076,149.219
C07987=1127.166,-13.688,-49.471,179.573,6.080,149.220
C07988=1127.162,-13.438,-49.484,179.574,6.085,149.220
C07989=1127.157,-13.189,-49.497,179.574,6.090,149.221
C07990=1127.151,-12.939,-49.509,179.575,6.095,149.222
C07991=1127.146,-12.690,-49.521,179.576,6.099,149.223
C07992=1127.140,-12.440,-49.535,179.576,6.104,149.224
C07993=1127.135,-12.191,-49.547,179.577,6.108,149.224
C07994=1127.130,-11.940,-49.559,179.578,6.113,149.225
C07995=1127.125,-11.691,-49.572,179.578,6.118,149.226
C07996=1127.120,-11.441,-49.585,179.579,6.122,149.227
C07997=1127.115,-11.192,-49.597,179.580,6.127,149.228
C07998=1127.110,-10.943,-49.610,179.581,6.131,149.228
C07999=1127.104,-10.692,-49.623,179.581,6.136,149.229
C08000=1127.099,-10.442,-49.635,179.582,6.141,149.230
C08001=1127.094,-10.193,-49.648,179.583,6.145,149.231
C08002=1127.089,-9.944,-49.660,179.583,6.150,149.232
C08003=1127.084,-9.694,-49.673,179.584,6.154,149.233
C08004=1127.079,-9.444,-49.686,179.585,6.159,149.233
C08005=1127.073,-9.195,-49.699,179.585,6.164,149.234
C08006=1127.068,-8.945,-49.711,179.586,6.168,149.235
C08007=1127.063,-8.696,-49.724,179.587,6.173,149.236
C08008=1127.058,-8.446,-49.737,179.587,6.177,149.237
C08009=1127.053,-8.196,-49.749,179.588,6.182,149.237
C08010=1127.047,-7.947,-49.763,179.589,6.186,149.238
C08011=1127.042,-7.697,-49.775,179.589,6.191,149.239
C08012=1127.038,-7.447,-49.788,179.590,6.196,149.240
C08013=1127.033,-7.198,-49.801,179.591,6.200,149.241
C08014=1127.028,-6.982,-49.812,179.591,6.204,149.241
C08015=1127.023,-6.768,-49.823,179.592,6.208,149.242
C08016=1127.019,-6.552,-49.834,179.592,6.212,149.243
C08017=1127.015,-6.336,-49.846,179.593,6.216,149.243
C08018=1127.010,-6.121,-49.856,179.594,6.220,149.244
C08019=1127.005,-5.905,-49.867,179.594,6.223,149.245
C08020=1127.001,-5.690,-49.879,179.595,6.228,149.245
C08021=1126.997,-5.474,-49.890,179.595,6.232,149.246
C08022=1126.991,-5.225,-49.902,179.596,6.236,149.247
C08023=1126.986,-4.976,-49.915,179.596,6.241,149.248
C08024=1126.981,-4.726,-49.929,179.597,6.246,149.249
C08025=1126.976,-4.476,-49.942,179.598,6.250,149.249
C08026=1126.971,-4.227,-49.955,179.598,6.255,149.250
C08027=1126.966,-3.977,-49.968,179.599,6.259,149.251
C08028=1126.961,-3.728,-49.981,179.599,6.263,149.252
C08029=1126.956,-3.478,-49.993,179.600,6.268,149.253
C08030=1126.950,-3.228,-50.007,179.600,6.272,149.254
C08031=1126.945,-2.979,-50.019,179.601,6.277,149.254
C08032=1126.940,-2.729,-50.032,179.602,6.281,149.255
C08033=1126.935,-2.479,-50.046,179.602,6.286,149.256
C08034=1126.930,-2.230,-50.059,179.603,6.291,149.257
C08035=1126.924,-1.981,-50.072,179.604,6.295,149.258
C08036=1126.920,-1.731,-50.085,179.604,6.299,149.258
C08037=1126.914,-1.481,-50.098,179.604,6.304,149.259
C08038=1126.909,-1.232,-50.111,179.605,6.309,149.260
C08039=1126.904,-0.982,-50.124,179.606,6.313,149.261
C08040=1126.899,-0.733,-50.138,179.606,6.318,149.262
C08041=1126.894,-0.483,-50.151,179.607,6.322,149.263
C08042=1126.888,-0.233,-50.164,179.607,6.326,149.263
C08043=1126.883,0.016,-50.177,179.608,6.331,149.264
C08044=1126.878,0.267,-50.190,179.608,6.335,149.265
C08045=1126.873,0.515,-50.203,179.609,6.340,149.266
C08046=1126.868,0.766,-50.217,179.609,6.345,149.267
C08047=1126.863,1.015,-50.230,179.610,6.349,149.267
C08048=1126.857,1.264,-50.242,179.610,6.353,149.268
C08049=1126.852,1.514,-50.256,179.611,6.358,149.269
C08050=1126.847,1.763,-50.269,179.611,6.362,149.270
C08051=1126.842,2.014,-50.283,179.612,6.367,149.271
C08052=1126.837,2.262,-50.296,179.613,6.372,149.272
C08053=1126.832,2.513,-50.309,179.613,6.375,149.273
C08054=1126.826,2.762,-50.323,179.613,6.380,149.273
C08055=1126.822,3.012,-50.336,179.614,6.385,149.274
C08056=1126.816,3.261,-50.350,179.614,6.390,149.275
C08057=1126.811,3.511,-50.362,179.615,6.394,149.276
C08058=1126.806,3.760,-50.376,179.615,6.398,149.277
C08059=1126.801,4.010,-50.389,179.616,6.403,149.278
C08060=1126.796,4.260,-50.403,179.616,6.407,149.278
C08061=1126.791,4.509,-50.416,179.617,6.412,149.279
C08062=1126.786,4.759,-50.429,179.618,6.417,149.280
C08063=1126.781,5.008,-50.443,179.618,6.420,149.281
C08064=1126.775,5.258,-50.456,179.618,6.425,149.282
C08065=1126.770,5.507,-50.470,179.619,6.430,149.283
C08066=1126.765,5.757,-50.483,179.620,6.434,149.284
C08067=1126.760,6.007,-50.496,179.620,6.438,149.284
C08068=1126.755,6.256,-50.510,179.620,6.443,149.285
C08069=1126.749,6.506,-50.523,179.621,6.448,149.286
C08070=1126.745,6.721,-50.535,179.621,6.451,149.287
C08071=1126.741,6.936,-50.547,179.621,6.455,149.288
C08072=1126.736,7.152,-50.559,179.622,6.460,149.288
C08073=1126.732,7.367,-50.571,179.622,6.463,149.289
C08074=1126.728,7.582,-50.582,179.622,6.467,149.290
C08075=1126.724,7.798,-50.594,179.623,6.471,149.291
C08076=1126.719,8.012,-50.605,179.623,6.475,149.291
C08077=1126.714,8.228,-50.618,179.624,6.479,149.292
C08078=1126.709,8.478,-50.631,179.624,6.484,149.293
C08079=1126.704,8.727,-50.644,179.625,6.488,149.294
C08080=1126.699,8.977,-50.658,179.626,6.493,149.294
C08081=1126.694,9.227,-50.672,179.627,6.498,149.295
C08082=1126.689,9.476,-50.685,179.628,6.503,149.296
C08083=1126.684,9.726,-50.699,179.628,6.507,149.297
C08084=1126.678,9.975,-50.712,179.630,6.512,149.298
C08085=1126.674,10.225,-50.726,179.630,6.516,149.298
C08086=1126.668,10.474,-50.740,179.631,6.522,149.299
C08087=1126.663,10.724,-50.754,179.632,6.526,149.300
C08088=1126.658,10.974,-50.767,179.633,6.531,149.301
C08089=1126.653,11.223,-50.781,179.634,6.535,149.301
C08090=1126.648,11.473,-50.795,179.634,6.540,149.302
C08091=1126.642,11.722,-50.809,179.636,6.545,149.303
C08092=1126.638,11.971,-50.822,179.637,6.550,149.304
C08093=1126.633,12.222,-50.836,179.638,6.554,149.305
C08094=1126.627,12.471,-50.850,179.638,6.559,149.305
C08095=1126.622,12.721,-50.864,179.639,6.563,149.306
C08096=1126.618,12.971,-50.877,179.640,6.569,149.307
C08097=1126.612,13.220,-50.891,179.641,6.573,149.308
C08098=1126.607,13.469,-50.905,179.642,6.578,149.308
C08099=1126.602,13.718,-50.919,179.643,6.582,149.309
C08100=1126.596,13.969,-50.933,179.644,6.587,149.310
C08101=1126.591,14.218,-50.947,179.645,6.591,149.311
C08102=1126.587,14.467,-50.960,179.646,6.596,149.312
C08103=1126.582,14.717,-50.975,179.647,6.601,149.312
C08104=1126.577,14.966,-50.989,179.647,6.606,149.313
C08105=1126.571,15.217,-51.002,179.648,6.610,149.314
C08106=1126.566,15.466,-51.016,179.649,6.614,149.314
C08107=1126.561,15.716,-51.031,179.650,6.619,149.315
C08108=1126.556,15.965,-51.045,179.651,6.623,149.316
C08109=1126.550,16.214,-51.059,179.652,6.629,149.317
C08110=1126.546,16.464,-51.072,179.653,6.633,149.317
C08111=1126.541,16.713,-51.087,179.654,6.637,149.318
C08112=1126.535,16.963,-51.100,179.655,6.642,149.319
C08113=1126.530,17.213,-51.114,179.656,6.646,149.320
C08114=1126.525,17.462,-51.128,179.657,6.651,149.320
C08115=1126.520,17.712,-51.143,179.657,6.655,149.321
C08116=1126.515,17.961,-51.157,179.659,6.661,149.322
C08117=1126.510,18.211,-51.171,179.660,6.665,149.322
C08118=1126.505,18.461,-51.185,179.661,6.670,149.323
C08119=1126.500,18.710,-51.199,179.662,6.674,149.324
C08120=1126.494,18.959,-51.213,179.663,6.678,149.325
C08121=1126.489,19.209,-51.228,179.663,6.683,149.325
C08122=1126.485,19.459,-51.242,179.664,6.687,149.326
C08123=1126.480,19.708,-51.256,179.666,6.692,149.327
C08124=1126.474,19.957,-51.270,179.667,6.697,149.328
C08125=1126.469,20.207,-51.284,179.668,6.701,149.328
C08126=1126.465,20.422,-51.296,179.668,6.705,149.329
C08127=1126.460,20.637,-51.309,179.670,6.709,149.329
C08128=1126.456,20.853,-51.321,179.670,6.712,149.330
C08129=1126.452,21.068,-51.334,179.671,6.717,149.331
C08130=1126.447,21.283,-51.345,179.672,6.720,149.331
C08131=1126.443,21.498,-51.359,179.673,6.725,149.332
C08132=1126.439,21.714,-51.370,179.674,6.729,149.332
C08133=1126.434,21.929,-51.383,179.674,6.732,149.333
C08134=1126.429,22.178,-51.397,179.676,6.736,149.334
C08135=1126.424,22.427,-51.412,179.677,6.741,149.334
C08136=1126.419,22.677,-51.426,179.677,6.745,149.335
C08137=1126.414,22.927,-51.440,179.679,6.751,149.336
C08138=1126.409,23.177,-51.454,179.680,6.755,149.336
C08139=1126.404,23.426,-51.469,179.681,6.759,149.337
C08140=1126.399,23.676,-51.484,179.682,6.763,149.338
C08141=1126.393,23.925,-51.498,179.683,6.768,149.338
C08142=1126.388,24.174,-51.513,179.684,6.772,149.339
C08143=1126.383,24.424,-51.527,179.685,6.777,149.340
C08144=1126.378,24.674,-51.541,179.686,6.781,149.341
C08145=1126.373,24.923,-51.555,179.687,6.785,149.341
C08146=1126.369,25.173,-51.570,179.688,6.790,149.342
C08147=1126.363,25.423,-51.585,179.689,6.794,149.343
C08148=1126.358,25.672,-51.599,179.690,6.798,149.343
C08149=1126.353,25.921,-51.614,179.692,6.804,149.344
C08150=1126.348,26.170,-51.628,179.692,6.808,149.345
C08151=1126.343,26.420,-51.643,179.693,6.813,149.345
C08152=1126.337,26.670,-51.658,179.694,6.817,149.346
C08153=1126.333,26.919,-51.673,179.695,6.821,149.347
C08154=1126.328,27.169,-51.687,179.696,6.825,149.347
C08155=1126.323,27.419,-51.701,179.697,6.830,149.348
C08156=1126.318,27.668,-51.716,179.698,6.834,149.349
C08157=1126.312,27.918,-51.731,179.700,6.838,149.349
C08158=1126.307,28.167,-51.745,179.701,6.843,149.350
C08159=1126.303,28.417,-51.760,179.702,6.847,149.351
C08160=1126.298,28.666,-51.775,179.703,6.851,149.351
C08161=1126.292,28.915,-51.790,179.704,6.856,149.352
C08162=1126.287,29.165,-51.804,179.705,6.860,149.353
C08163=1126.282,29.414,-51.818,179.706,6.864,149.353
C08164=1126.277,29.664,-51.834,179.708,6.869,149.354
C08165=1126.272,29.914,-51.848,179.709,6.874,149.354
C08166=1126.267,30.163,-51.863,179.710,6.878,149.355
C08167=1126.262,30.412,-51.877,179.711,6.882,149.356
C08168=1126.257,30.662,-51.893,179.712,6.887,149.356
C08169=1126.252,30.911,-51.907,179.713,6.891,149.357
C08170=1126.247,31.161,-51.922,179.714,6.895,149.358
C08171=1126.241,31.411,-51.937,179.715,6.900,149.358
C08172=1126.237,31.660,-51.952,179.716,6.904,149.359
C08173=1126.232,31.909,-51.966,179.717,6.908,149.360
C08174=1126.226,32.159,-51.982,179.718,6.913,149.360
C08175=1126.221,32.408,-51.996,179.720,6.916,149.361
C08176=1126.216,32.658,-52.012,179.721,6.921,149.361
C08177=1126.211,32.908,-52.026,179.722,6.925,149.362
C08178=1126.207,33.157,-52.042,179.723,6.929,149.363
C08179=1126.202,33.407,-52.057,179.724,6.934,149.363
C08180=1126.197,33.656,-52.071,179.725,6.938,149.364
C08181=1126.191,33.906,-52.087,179.726,6.942,149.365
C08182=1126.187,34.121,-52.099,179.728,6.946,149.365
C08183=1126.183,34.335,-52.112,179.728,6.950,149.366
C08184=1126.178,34.550,-52.125,179.730,6.954,149.366
C08185=1126.174,34.766,-52.139,179.730,6.957,149.367
C08186=1126.170,34.981,-52.152,179.732,6.961,149.367
C08187=1126.165,35.196,-52.165,179.732,6.965,149.368
C08188=1126.161,35.411,-52.177,179.733,6.968,149.368
C08189=1126.157,35.627,-52.190,179.734,6.972,149.369
C08190=1126.151,35.876,-52.205,179.735,6.976,149.369
C08191=1126.147,36.125,-52.220,179.737,6.980,149.370
C08192=1126.141,36.375,-52.236,179.738,6.985,149.371
C08193=1126.136,36.625,-52.250,179.739,6.989,149.371
C08194=1126.131,36.874,-52.266,179.740,6.993,149.372
C08195=1126.126,37.123,-52.281,179.741,6.998,149.373
C08196=1126.121,37.372,-52.296,179.742,7.002,149.373
C08197=1126.116,37.622,-52.311,179.743,7.006,149.374
C08198=1126.111,37.872,-52.327,179.745,7.010,149.374
C08199=1126.107,38.121,-52.342,179.746,7.014,149.375
C08200=1126.101,38.371,-52.357,179.747,7.018,149.375
C08201=1126.096,38.620,-52.373,179.748,7.023,149.376
C08202=1126.091,38.870,-52.387,179.749,7.027,149.377
C08203=1126.086,39.119,-52.403,179.750,7.031,149.377
C08204=1126.081,39.368,-52.418,179.752,7.035,149.378
C08205=1126.076,39.618,-52.434,179.753,7.040,149.378
C08206=1126.071,39.868,-52.449,179.754,7.044,149.379
C08207=1126.066,40.117,-52.464,179.755,7.048,149.380
C08208=1126.060,40.367,-52.479,179.757,7.052,149.380
C08209=1126.056,40.616,-52.494,179.758,7.056,149.381
C08210=1126.051,40.866,-52.510,179.759,7.061,149.381
C08211=1126.046,41.116,-52.526,179.760,7.065,149.382
C08212=1126.041,41.365,-52.541,179.761,7.069,149.382
C08213=1126.036,41.614,-52.556,179.762,7.073,149.383
C08214=1126.030,41.863,-52.572,179.764,7.078,149.384
C08215=1126.026,42.113,-52.587,179.765,7.081,149.384
C08216=1126.021,42.363,-52.603,179.766,7.086,149.385
C08217=1126.015,42.612,-52.618,179.767,7.090,149.385
C08218=1126.011,42.861,-52.633,179.769,7.094,149.386
C08219=1126.005,43.111,-52.649,179.770,7.098,149.387
C08220=1126.000,43.361,-52.665,179.771,7.103,149.387
C08221=1125.996,43.610,-52.680,179.772,7.107,149.388
C08222=1125.990,43.859,-52.695,179.774,7.111,149.388
C08223=1125.985,44.109,-52.711,179.775,7.115,149.389
C08224=1125.981,44.358,-52.726,179.776,7.119,149.389
C08225=1125.976,44.608,-52.742,179.777,7.123,149.390
C08226=1125.970,44.857,-52.757,179.778,7.128,149.391
C08227=1125.965,45.107,-52.773,179.780,7.132,149.391
C08228=1125.961,45.356,-52.788,179.781,7.136,149.392
C08229=1125.956,45.605,-52.805,179.782,7.140,149.392
C08230=1125.950,45.855,-52.820,179.784,7.144,149.393
C08231=1125.946,46.105,-52.836,179.785,7.148,149.393
C08232=1125.940,46.354,-52.852,179.786,7.152,149.394
C08233=1125.936,46.603,-52.867,179.787,7.157,149.394
C08234=1125.931,46.853,-52.883,179.788,7.161,149.395
C08235=1125.925,47.103,-52.898,179.790,7.165,149.396
C08236=1125.920,47.351,-52.915,179.791,7.169,149.396
C08237=1125.915,47.602,-52.931,179.793,7.173,149.397
C08238=1125.911,47.816,-52.944,179.793,7.177,149.397
C08239=1125.907,48.031,-52.957,179.795,7.181,149.398
C08240=1125.903,48.246,-52.971,179.796,7.184,149.398
C08241=1125.898,48.461,-52.984,179.796,7.187,149.399
C08242=1125.894,48.676,-52.998,179.798,7.191,149.399
C08243=1125.890,48.891,-53.011,179.798,7.194,149.400
C08244=1125.885,49.107,-53.025,179.800,7.198,149.400
C08245=1125.881,49.321,-53.039,179.801,7.201,149.401
C08246=1125.876,49.571,-53.055,179.802,7.206,149.401
C08247=1125.871,49.821,-53.071,179.804,7.209,149.402
C08248=1125.866,50.069,-53.086,179.805,7.214,149.402
C08249=1125.862,50.319,-53.102,179.806,7.218,149.403
C08250=1125.856,50.569,-53.118,179.807,7.222,149.403
C08251=1125.851,50.817,-53.134,179.809,7.226,149.404
C08252=1125.846,51.067,-53.150,179.810,7.230,149.404
C08253=1125.841,51.317,-53.166,179.812,7.234,149.405
C08254=1125.837,51.566,-53.182,179.813,7.238,149.405
C08255=1125.831,51.816,-53.198,179.814,7.242,149.406
C08256=1125.827,52.065,-53.215,179.815,7.247,149.407
C08257=1125.821,52.315,-53.230,179.817,7.251,149.407
C08258=1125.816,52.564,-53.246,179.818,7.255,149.408
C08259=1125.811,52.814,-53.263,179.819,7.259,149.408
C08260=1125.806,53.063,-53.278,179.821,7.263,149.409
C08261=1125.802,53.312,-53.295,179.822,7.267,149.409
C08262=1125.796,53.562,-53.310,179.823,7.271,149.410
C08263=1125.792,53.811,-53.327,179.825,7.275,149.410
C08264=1125.786,54.061,-53.343,179.826,7.279,149.411
C08265=1125.781,54.309,-53.359,179.827,7.283,149.411
C08266=1125.776,54.560,-53.375,179.828,7.287,149.412
C08267=1125.771,54.808,-53.391,179.829,7.291,149.412
C08268=1125.767,55.058,-53.407,179.831,7.295,149.413
C08269=1125.761,55.307,-53.423,179.832,7.299,149.413
C08270=1125.757,55.557,-53.439,179.833,7.303,149.414
C08271=1125.752,55.806,-53.456,179.835,7.307,149.414
C08272=1125.747,56.056,-53.472,179.836,7.311,149.415
C08273=1125.742,56.305,-53.488,179.837,7.315,149.416
C08274=1125.737,56.555,-53.504,179.839,7.319,149.416
C08275=1125.731,56.804,-53.521,179.840,7.324,149.417
C08276=1125.727,57.054,-53.538,179.842,7.328,149.417
C08277=1125.721,57.303,-53.553,179.843,7.332,149.418
C08278=1125.717,57.553,-53.570,179.844,7.336,149.418
C08279=1125.711,57.802,-53.585,179.846,7.340,149.419
C08280=1125.707,58.051,-53.602,179.847,7.344,149.419
C08281=1125.702,58.300,-53.618,179.848,7.348,149.420
C08282=1125.697,58.550,-53.634,179.850,7.352,149.420
C08283=1125.691,58.799,-53.651,179.851,7.356,149.421
C08284=1125.687,59.049,-53.668,179.853,7.360,149.421
C08285=1125.682,59.298,-53.685,179.854,7.364,149.422
C08286=1125.677,59.548,-53.700,179.855,7.368,149.422
C08287=1125.672,59.797,-53.717,179.856,7.373,149.423
C08288=1125.667,60.046,-53.733,179.858,7.376,149.423
C08289=1125.662,60.297,-53.750,179.860,7.380,149.424
C08290=1125.657,60.545,-53.766,179.860,7.384,149.424
C08291=1125.652,60.795,-53.783,179.862,7.388,149.425
C08292=1125.648,61.044,-53.799,179.863,7.392,149.425
C08293=1125.642,61.293,-53.816,179.864,7.396,149.426
C08294=1125.638,61.508,-53.830,179.866,7.400,149.426
C08295=1125.634,61.724,-53.845,179.867,7.403,149.427
C08296=1125.630,61.938,-53.859,179.868,7.407,149.427
C08297=1125.625,62.153,-53.873,179.869,7.410,149.428
C08298=1125.621,62.368,-53.887,179.870,7.413,149.428
C08299=1125.616,62.583,-53.902,179.872,7.417,149.428
C08300=1125.613,62.798,-53.916,179.873,7.420,149.429
C08301=1125.608,63.013,-53.930,179.874,7.424,149.429
C08302=1125.603,63.262,-53.947,179.876,7.428,149.430
C08303=1125.599,63.512,-53.963,179.876,7.432,149.430
C08304=1125.594,63.761,-53.980,179.878,7.435,149.431
C08305=1125.588,64.011,-53.996,179.879,7.440,149.431
C08306=1125.584,64.260,-54.013,179.881,7.444,149.432
C08307=1125.578,64.509,-54.029,179.882,7.448,149.432
C08308=1125.573,64.759,-54.046,179.883,7.452,149.433
C08309=1125.569,65.009,-54.063,179.885,7.456,149.433
C08310=1125.564,65.257,-54.079,179.886,7.460,149.434
C08311=1125.558,65.507,-54.097,179.888,7.464,149.434
C08312=1125.554,65.757,-54.113,179.889,7.468,149.435
C08313=1125.549,66.005,-54.130,179.891,7.472,149.435
C08314=1125.544,66.255,-54.147,179.892,7.476,149.436
C08315=1125.539,66.505,-54.164,179.893,7.480,149.436
C08316=1125.534,66.754,-54.181,179.895,7.484,149.437
C08317=1125.529,67.003,-54.197,179.896,7.488,149.437
C08318=1125.524,67.253,-54.214,179.898,7.492,149.438
C08319=1125.519,67.502,-54.231,179.899,7.496,149.438
C08320=1125.514,67.751,-54.247,179.901,7.500,149.439
C08321=1125.509,68.000,-54.265,179.902,7.504,149.439
C08322=1125.505,68.250,-54.282,179.903,7.508,149.440
C08323=1125.500,68.500,-54.299,179.905,7.512,149.440
C08324=1125.494,68.748,-54.316,179.907,7.516,149.441
C08325=1125.490,68.998,-54.332,179.908,7.520,149.441
C08326=1125.485,69.248,-54.350,179.909,7.523,149.442
C08327=1125.480,69.497,-54.366,179.910,7.527,149.442
C08328=1125.474,69.746,-54.383,179.911,7.531,149.443
C08329=1125.470,69.995,-54.401,179.913,7.535,149.443
C08330=1125.465,70.245,-54.418,179.914,7.539,149.444
C08331=1125.461,70.495,-54.434,179.916,7.543,149.444
C08332=1125.455,70.744,-54.452,179.917,7.547,149.445
C08333=1125.450,70.993,-54.468,179.919,7.551,149.445
C08334=1125.445,71.242,-54.486,179.920,7.555,149.445
C08335=1125.440,71.492,-54.503,179.922,7.559,149.446
C08336=1125.436,71.742,-54.520,179.923,7.563,149.447
C08337=1125.430,71.991,-54.537,179.925,7.567,149.447
C08338=1125.426,72.239,-54.554,179.926,7.571,149.447
C08339=1125.420,72.489,-54.571,179.927,7.576,149.448
C08340=1125.416,72.739,-54.588,179.929,7.579,149.448
C08341=1125.411,72.989,-54.605,179.930,7.583,149.449
C08342=1125.407,73.237,-54.623,179.932,7.587,149.449
C08343=1125.401,73.487,-54.640,179.933,7.592,149.450
C08344=1125.396,73.736,-54.657,179.935,7.595,149.450
C08345=1125.391,73.985,-54.674,179.936,7.599,149.451
C08346=1125.386,74.235,-54.692,179.938,7.603,149.451
C08347=1125.381,74.485,-54.709,179.939,7.608,149.452
C08348=1125.377,74.734,-54.726,179.941,7.611,149.452
C08349=1125.372,74.983,-54.744,179.942,7.615,149.453
C08350=1125.367,75.198,-54.759,179.943,7.618,149.453
C08351=1125.363,75.412,-54.773,179.944,7.622,149.454
C08352=1125.359,75.627,-54.788,179.946,7.625,149.454
C08353=1125.355,75.842,-54.803,179.947,7.629,149.454
C08354=1125.350,76.057,-54.818,179.948,7.632,149.455
C08355=1125.346,76.272,-54.833,179.949,7.636,149.455
C08356=1125.342,76.487,-54.848,179.951,7.639,149.456
C08357=1125.337,76.701,-54.863,179.952,7.642,149.456
C08358=1125.333,76.951,-54.880,179.953,7.646,149.457
C08359=1125.328,77.200,-54.898,179.954,7.650,149.457
C08360=1125.323,77.450,-54.915,179.955,7.653,149.458
C08361=1125.318,77.699,-54.932,179.956,7.657,149.458
C08362=1125.313,77.949,-54.950,179.957,7.661,149.459
C08363=1125.308,78.198,-54.968,179.958,7.665,149.459
C08364=1125.303,78.447,-54.986,179.958,7.668,149.460
C08365=1125.299,78.696,-55.002,179.960,7.672,149.460
C08366=1125.294,78.946,-55.020,179.961,7.676,149.461
C08367=1125.289,79.195,-55.038,179.962,7.680,149.462
C08368=1125.284,79.444,-55.056,179.963,7.683,149.462
C08369=1125.279,79.694,-55.072,179.964,7.687,149.463
C08370=1125.274,79.943,-55.090,179.965,7.691,149.463
C08371=1125.269,80.193,-55.107,179.966,7.694,149.464
C08372=1125.264,80.442,-55.125,179.967,7.698,149.464
C08373=1125.259,80.691,-55.143,179.968,7.702,149.465
C08374=1125.254,80.940,-55.160,179.969,7.705,149.465
C08375=1125.249,81.189,-55.178,179.970,7.709,149.466
C08376=1125.244,81.438,-55.196,179.972,7.713,149.466
C08377=1125.239,81.688,-55.213,179.973,7.717,149.467
C08378=1125.234,81.937,-55.231,179.974,7.721,149.468
C08379=1125.229,82.187,-55.249,179.975,7.724,149.468
C08380=1125.225,82.436,-55.266,179.976,7.728,149.468
C08381=1125.220,82.685,-55.284,179.977,7.732,149.469
C08382=1125.215,82.934,-55.302,179.978,7.735,149.469
C08383=1125.211,83.185,-55.319,179.979,7.740,149.470
C08384=1125.206,83.434,-55.337,179.981,7.743,149.471
C08385=1125.201,83.683,-55.355,179.982,7.747,149.471
C08386=1125.196,83.932,-55.373,179.983,7.751,149.472
C08387=1125.191,84.182,-55.390,179.985,7.755,149.472
C08388=1125.186,84.431,-55.408,179.986,7.759,149.473
C08389=1125.181,84.680,-55.426,179.987,7.762,149.473
C08390=1125.177,84.929,-55.444,179.988,7.766,149.474
C08391=1125.171,85.179,-55.461,179.990,7.770,149.474
C08392=1125.166,85.428,-55.479,179.991,7.773,149.475
C08393=1125.162,85.678,-55.497,179.992,7.777,149.475
C08394=1125.157,85.927,-55.515,179.993,7.782,149.476
C08395=1125.152,86.176,-55.533,179.995,7.786,149.476
C08396=1125.147,86.425,-55.551,179.996,7.789,149.477
C08397=1125.142,86.675,-55.568,179.997,7.793,149.477
C08398=1125.137,86.924,-55.586,179.999,7.797,149.478
C08399=1125.132,87.173,-55.604,-180.000,7.801,149.478
C08400=1125.127,87.423,-55.622,-179.999,7.805,149.479
C08401=1125.123,87.672,-55.640,-179.997,7.809,149.479
C08402=1125.118,87.922,-55.658,-179.996,7.812,149.480
C08403=1125.113,88.171,-55.676,-179.995,7.816,149.480
C08404=1125.108,88.420,-55.694,-179.993,7.820,149.481
C08405=1125.103,88.669,-55.712,-179.992,7.824,149.481
C08406=1125.099,88.884,-55.728,-179.991,7.827,149.481
C08407=1125.095,89.098,-55.743,-179.989,7.831,149.482
C08408=1125.090,89.313,-55.758,-179.988,7.834,149.482
C08409=1125.086,89.528,-55.774,-179.987,7.837,149.483
C08410=1125.081,89.743,-55.790,-179.985,7.841,149.483
C08411=1125.077,89.958,-55.805,-179.984,7.844,149.483
C08412=1125.073,90.172,-55.821,-179.983,7.848,149.484
C08413=1125.069,90.387,-55.836,-179.982,7.851,149.484
C08414=1125.064,90.636,-55.854,-179.980,7.855,149.485
C08415=1125.060,90.886,-55.873,-179.979,7.859,149.485
C08416=1125.055,91.135,-55.891,-179.977,7.863,149.486
C08417=1125.050,91.384,-55.909,-179.975,7.866,149.486
C08418=1125.045,91.633,-55.928,-179.974,7.870,149.486
C08419=1125.040,91.883,-55.946,-179.972,7.874,149.487
C08420=1125.035,92.132,-55.964,-179.971,7.878,149.487
C08421=1125.031,92.382,-55.982,-179.969,7.882,149.488
C08422=1125.026,92.631,-56.000,-179.967,7.886,149.488
C08423=1125.021,92.880,-56.018,-179.966,7.890,149.489
C08424=1125.016,93.129,-56.036,-179.964,7.894,149.489
C08425=1125.011,93.379,-56.055,-179.963,7.898,149.489
C08426=1125.006,93.628,-56.073,-179.961,7.901,149.490
C08427=1125.001,93.877,-56.091,-179.959,7.905,149.490
C08428=1124.996,94.126,-56.109,-179.958,7.909,149.491
C08429=1124.991,94.375,-56.127,-179.956,7.913,149.491
C08430=1124.986,94.626,-56.146,-179.955,7.917,149.492
C08431=1124.982,94.874,-56.165,-179.953,7.921,149.492
C08432=1124.977,95.123,-56.183,-179.951,7.925,149.492
C08433=1124.972,95.373,-56.201,-179.950,7.929,149.493
C08434=1124.968,95.622,-56.219,-179.948,7.933,149.493
C08435=1124.962,95.871,-56.239,-179.946,7.937,149.494
C08436=1124.957,96.120,-56.257,-179.944,7.941,149.494
C08437=1124.952,96.370,-56.275,-179.942,7.945,149.494
C08438=1124.948,96.619,-56.294,-179.941,7.949,149.495
C08439=1124.943,96.868,-56.312,-179.939,7.952,149.495
C08440=1124.938,97.118,-56.330,-179.937,7.956,149.496
C08441=1124.934,97.367,-56.349,-179.936,7.960,149.496
C08442=1124.928,97.616,-56.368,-179.934,7.965,149.496
C08443=1124.923,97.865,-56.386,-179.932,7.968,149.497
C08444=1124.919,98.115,-56.405,-179.930,7.972,149.497
C08445=1124.914,98.364,-56.423,-179.928,7.976,149.498
C08446=1124.909,98.613,-56.441,-179.926,7.980,149.498
C08447=1124.905,98.863,-56.461,-179.925,7.984,149.498
C08448=1124.899,99.112,-56.479,-179.923,7.988,149.499
C08449=1124.895,99.361,-56.498,-179.921,7.992,149.499
C08450=1124.890,99.611,-56.516,-179.919,7.996,149.499
C08451=1124.885,99.859,-56.535,-179.917,8.000,149.500
C08452=1124.880,100.109,-56.553,-179.915,8.004,149.500
C08453=1124.875,100.358,-56.573,-179.913,8.008,149.500
C08454=1124.870,100.607,-56.591,-179.911,8.012,149.501
C08455=1124.866,100.856,-56.610,-179.909,8.015,149.501
C08456=1124.861,101.106,-56.629,-179.907,8.020,149.501
C08457=1124.856,101.355,-56.647,-179.905,8.023,149.502
C08458=1124.851,101.605,-56.666,-179.903,8.027,149.502
C08459=1124.846,101.853,-56.685,-179.901,8.031,149.502
C08460=1124.841,102.103,-56.704,-179.899,8.035,149.503
C08461=1124.837,102.352,-56.723,-179.897,8.039,149.503
C08462=1124.832,102.567,-56.739,-179.895,8.043,149.503
C08463=1124.828,102.781,-56.755,-179.893,8.046,149.504
C08464=1124.823,102.996,-56.771,-179.892,8.049,149.504
C08465=1124.820,103.211,-56.788,-179.890,8.052,149.504
C08466=1124.815,103.426,-56.804,-179.888,8.056,149.504
C08467=1124.812,103.640,-56.820,-179.887,8.059,149.505
C08468=1124.807,103.854,-56.837,-179.885,8.063,149.505
C08469=1124.804,104.070,-56.852,-179.883,8.066,149.505
C08470=1124.798,104.318,-56.872,-179.881,8.070,149.506
C08471=1124.794,104.568,-56.891,-179.878,8.074,149.506
C08472=1124.789,104.816,-56.910,-179.876,8.078,149.506
C08473=1124.784,105.066,-56.928,-179.875,8.082,149.506
C08474=1124.779,105.315,-56.948,-179.872,8.086,149.507
C08475=1124.775,105.564,-56.967,-179.870,8.089,149.507
C08476=1124.770,105.813,-56.986,-179.867,8.094,149.507
C08477=1124.765,106.064,-57.005,-179.866,8.098,149.508
C08478=1124.760,106.312,-57.024,-179.864,8.101,149.508
C08479=1124.755,106.562,-57.043,-179.861,8.105,149.508
C08480=1124.751,106.810,-57.062,-179.859,8.109,149.508
C08481=1124.746,107.060,-57.082,-179.857,8.114,149.509
C08482=1124.741,107.309,-57.101,-179.855,8.117,149.509
C08483=1124.736,107.559,-57.119,-179.852,8.121,149.509
C08484=1124.731,107.807,-57.139,-179.850,8.125,149.509
C08485=1124.726,108.057,-57.158,-179.847,8.129,149.509
C08486=1124.722,108.306,-57.177,-179.845,8.133,149.510
C08487=1124.717,108.555,-57.197,-179.843,8.137,149.510
C08488=1124.712,108.804,-57.216,-179.840,8.140,149.510
C08489=1124.708,109.053,-57.235,-179.838,8.144,149.510
C08490=1124.703,109.303,-57.255,-179.836,8.148,149.511
C08491=1124.698,109.552,-57.274,-179.834,8.152,149.511
C08492=1124.693,109.801,-57.294,-179.831,8.156,149.511
C08493=1124.688,110.050,-57.312,-179.829,8.159,149.511
C08494=1124.683,110.299,-57.332,-179.826,8.164,149.511
C08495=1124.679,110.549,-57.352,-179.824,8.168,149.512
C08496=1124.673,110.798,-57.371,-179.821,8.171,149.512
C08497=1124.669,111.047,-57.390,-179.819,8.175,149.512
C08498=1124.664,111.296,-57.409,-179.817,8.178,149.512
C08499=1124.659,111.545,-57.429,-179.815,8.182,149.513
C08500=1124.655,111.795,-57.449,-179.814,8.186,149.513
C08501=1124.649,112.044,-57.468,-179.812,8.189,149.513
C08502=1124.644,112.293,-57.487,-179.810,8.193,149.513
C08503=1124.640,112.543,-57.507,-179.808,8.196,149.514
C08504=1124.635,112.791,-57.527,-179.806,8.200,149.514
C08505=1124.631,113.041,-57.546,-179.804,8.204,149.514
C08506=1124.625,113.289,-57.565,-179.802,8.207,149.515
C08507=1124.621,113.539,-57.585,-179.800,8.210,149.515
C08508=1124.616,113.789,-57.605,-179.799,8.214,149.515
C08509=1124.610,114.037,-57.624,-179.797,8.217,149.515
C08510=1124.607,114.286,-57.644,-179.795,8.221,149.516
C08511=1124.602,114.536,-57.664,-179.793,8.224,149.516
C08512=1124.597,114.785,-57.683,-179.790,8.228,149.516
C08513=1124.592,115.034,-57.702,-179.789,8.232,149.517
C08514=1124.588,115.283,-57.723,-179.787,8.235,149.517
C08515=1124.583,115.533,-57.742,-179.785,8.238,149.517
C08516=1124.577,115.781,-57.762,-179.783,8.241,149.517
C08517=1124.573,116.031,-57.781,-179.782,8.245,149.518
C08518=1124.569,116.246,-57.799,-179.780,8.249,149.518
C08519=1124.564,116.460,-57.816,-179.778,8.252,149.518
C08520=1124.560,116.674,-57.833,-179.777,8.254,149.518
C08521=1124.557,116.889,-57.850,-179.775,8.257,149.519
C08522=1124.552,117.103,-57.866,-179.773,8.260,149.519
C08523=1124.548,117.318,-57.884,-179.772,8.263,149.519
C08524=1124.544,117.532,-57.901,-179.770,8.266,149.519
C08525=1124.540,117.747,-57.918,-179.768,8.269,149.519
C08526=1124.536,117.997,-57.938,-179.767,8.272,149.520
C08527=1124.530,118.245,-57.958,-179.765,8.276,149.520
C08528=1124.526,118.494,-57.977,-179.763,8.279,149.520
C08529=1124.521,118.744,-57.997,-179.761,8.283,149.520
C08530=1124.517,118.993,-58.017,-179.759,8.286,149.521
C08531=1124.511,119.242,-58.037,-179.758,8.289,149.521
C08532=1124.507,119.491,-58.057,-179.756,8.293,149.521
C08533=1124.502,119.740,-58.077,-179.754,8.297,149.522
C08534=1124.498,119.989,-58.097,-179.752,8.300,149.522
C08535=1124.493,120.239,-58.117,-179.750,8.304,149.522
C08536=1124.488,120.488,-58.138,-179.748,8.306,149.522
C08537=1124.482,120.737,-58.157,-179.746,8.310,149.522
C08538=1124.478,120.986,-58.177,-179.745,8.314,149.523
C08539=1124.473,121.235,-58.197,-179.743,8.317,149.523
C08540=1124.469,121.484,-58.217,-179.741,8.320,149.523
C08541=1124.464,121.734,-58.237,-179.739,8.323,149.524
C08542=1124.459,121.982,-58.257,-179.737,8.327,149.524
C08543=1124.454,122.232,-58.277,-179.735,8.331,149.524
C08544=1124.450,122.481,-58.297,-179.734,8.333,149.524
C08545=1124.445,122.730,-58.318,-179.732,8.337,149.525
C08546=1124.440,122.980,-58.338,-179.730,8.340,149.525
C08547=1124.435,123.229,-58.358,-179.728,8.344,149.525
C08548=1124.431,123.477,-58.378,-179.727,8.347,149.526
C08549=1124.426,123.727,-58.398,-179.725,8.351,149.526
C08550=1124.421,123.975,-58.418,-179.723,8.354,149.526
C08551=1124.416,124.225,-58.438,-179.721,8.357,149.526
C08552=1124.411,124.474,-58.459,-179.720,8.361,149.527
C08553=1124.407,124.723,-58.479,-179.717,8.364,149.527
C08554=1124.402,124.972,-58.499,-179.715,8.368,149.527
C08555=1124.398,125.222,-58.519,-179.714,8.370,149.527
C08556=1124.392,125.471,-58.540,-179.712,8.374,149.528
C08557=1124.388,125.720,-58.560,-179.710,8.378,149.528
C08558=1124.383,125.969,-58.580,-179.709,8.380,149.528
C08559=1124.379,126.218,-58.600,-179.707,8.384,149.528
C08560=1124.374,126.468,-58.621,-179.705,8.387,149.529
C08561=1124.369,126.716,-58.641,-179.704,8.391,149.529
C08562=1124.364,126.965,-58.661,-179.702,8.394,149.529
C08563=1124.359,127.214,-58.681,-179.700,8.398,149.530
C08564=1124.354,127.464,-58.702,-179.698,8.400,149.530
C08565=1124.350,127.713,-58.723,-179.697,8.404,149.530
C08566=1124.345,127.961,-58.743,-179.694,8.408,149.530
C08567=1124.340,128.211,-58.764,-179.693,8.410,149.531
C08568=1124.335,128.460,-58.784,-179.691,8.414,149.531
C08569=1124.331,128.709,-58.804,-179.689,8.418,149.531
C08570=1124.326,128.959,-58.825,-179.688,8.420,149.532
C08571=1124.321,129.207,-58.846,-179.686,8.424,149.532
C08572=1124.317,129.456,-58.866,-179.684,8.428,149.532
C08573=1124.312,129.706,-58.887,-179.683,8.430,149.532
C08574=1124.308,129.920,-58.905,-179.681,8.433,149.533
C08575=1124.304,130.135,-58.921,-179.679,8.437,149.533
C08576=1124.300,130.349,-58.939,-179.678,8.439,149.533
C08577=1124.296,130.564,-58.957,-179.676,8.442,149.533
C08578=1124.291,130.778,-58.975,-179.675,8.445,149.534
C08579=1124.288,130.992,-58.993,-179.673,8.448,149.534
C08580=1124.284,131.207,-59.010,-179.672,8.451,149.534
C08581=1124.279,131.421,-59.028,-179.671,8.453,149.534
C08582=1124.275,131.670,-59.049,-179.669,8.457,149.535
C08583=1124.270,131.919,-59.069,-179.667,8.460,149.535
C08584=1124.265,132.168,-59.090,-179.666,8.463,149.535
C08585=1124.261,132.417,-59.111,-179.664,8.467,149.536
C08586=1124.256,132.667,-59.132,-179.662,8.470,149.536
C08587=1124.252,132.916,-59.152,-179.661,8.474,149.536
C08588=1124.246,133.165,-59.173,-179.659,8.477,149.536
C08589=1124.242,133.414,-59.194,-179.657,8.480,149.537
C08590=1124.237,133.663,-59.215,-179.656,8.484,149.537
C08591=1124.232,133.912,-59.235,-179.654,8.486,149.537
C08592=1124.227,134.161,-59.256,-179.652,8.490,149.538
C08593=1124.223,134.410,-59.276,-179.650,8.494,149.538
C08594=1124.218,134.660,-59.297,-179.649,8.496,149.538
C08595=1124.213,134.909,-59.318,-179.647,8.500,149.538
C08596=1124.208,135.157,-59.339,-179.646,8.503,149.539
C08597=1124.204,135.406,-59.360,-179.644,8.506,149.539
C08598=1124.199,135.655,-59.381,-179.642,8.509,149.539
C08599=1124.195,135.905,-59.401,-179.641,8.513,149.540
C08600=1124.190,136.154,-59.422,-179.639,8.517,149.540
C08601=1124.185,136.403,-59.443,-179.638,8.520,149.540
C08602=1124.180,136.652,-59.464,-179.636,8.523,149.541
C08603=1124.176,136.901,-59.485,-179.634,8.526,149.541
C08604=1124.171,137.150,-59.506,-179.632,8.530,149.541
C08605=1124.166,137.399,-59.526,-179.631,8.532,149.542
C08606=1124.161,137.648,-59.548,-179.629,8.536,149.542
C08607=1124.157,137.898,-59.569,-179.627,8.540,149.542
C08608=1124.152,138.147,-59.589,-179.626,8.543,149.543
C08609=1124.147,138.396,-59.610,-179.624,8.546,149.543
C08610=1124.143,138.644,-59.632,-179.623,8.549,149.543
C08611=1124.138,138.894,-59.652,-179.621,8.553,149.544
C08612=1124.133,139.143,-59.673,-179.620,8.556,149.544
C08613=1124.129,139.391,-59.695,-179.618,8.560,149.544
C08614=1124.124,139.641,-59.716,-179.617,8.562,149.544
C08615=1124.119,139.890,-59.737,-179.615,8.566,149.545
C08616=1124.115,140.139,-59.758,-179.614,8.569,149.545
C08617=1124.110,140.388,-59.779,-179.612,8.573,149.545
C08618=1124.104,140.637,-59.800,-179.610,8.575,149.546
C08619=1124.101,140.886,-59.821,-179.609,8.579,149.546
C08620=1124.096,141.135,-59.842,-179.607,8.583,149.546
C08621=1124.090,141.385,-59.863,-179.606,8.586,149.547
C08622=1124.086,141.633,-59.884,-179.604,8.589,149.547
C08623=1124.081,141.882,-59.905,-179.603,8.592,149.547
C08624=1124.077,142.132,-59.927,-179.601,8.596,149.548
C08625=1124.072,142.381,-59.948,-179.600,8.599,149.548
C08626=1124.068,142.629,-59.969,-179.598,8.603,149.549
C08627=1124.062,142.879,-59.990,-179.596,8.606,149.549
C08628=1124.058,143.128,-60.012,-179.595,8.609,149.549
C08629=1124.054,143.377,-60.033,-179.593,8.612,149.549
C08630=1124.049,143.592,-60.051,-179.592,8.615,149.550
C08631=1124.046,143.805,-60.070,-179.591,8.618,149.550
C08632=1124.041,144.020,-60.088,-179.589,8.621,149.550
C08633=1124.037,144.234,-60.105,-179.588,8.624,149.551
C08634=1124.033,144.448,-60.125,-179.587,8.626,149.551
C08635=1124.029,144.663,-60.143,-179.586,8.630,149.551
C08636=1124.026,144.877,-60.161,-179.585,8.632,149.552
C08637=1124.021,145.092,-60.180,-179.583,8.635,149.552
C08638=1124.016,145.340,-60.201,-179.580,8.639,149.552
C08639=1124.012,145.589,-60.222,-179.578,8.644,149.552
C08640=1124.008,145.839,-60.244,-179.576,8.647,149.553
C08641=1124.002,146.088,-60.265,-179.573,8.651,149.553
C08642=1123.997,146.337,-60.287,-179.571,8.655,149.553
C08643=1123.993,146.585,-60.308,-179.568,8.659,149.553
C08644=1123.988,146.835,-60.330,-179.566,8.663,149.554
C08645=1123.984,147.084,-60.351,-179.563,8.666,149.554
C08646=1123.979,147.332,-60.372,-179.560,8.671,149.554
C08647=1123.974,147.582,-60.394,-179.558,8.674,149.554
C08648=1123.970,147.831,-60.415,-179.555,8.678,149.554
C08649=1123.965,148.079,-60.437,-179.553,8.682,149.554
C08650=1123.960,148.329,-60.459,-179.550,8.686,149.555
C08651=1123.955,148.578,-60.480,-179.548,8.689,149.555
C08652=1123.950,148.827,-60.502,-179.545,8.694,149.555
C08653=1123.946,149.076,-60.524,-179.543,8.697,149.555
C08654=1123.941,149.325,-60.545,-179.540,8.701,149.555
C08655=1123.937,149.575,-60.567,-179.538,8.704,149.555
C08656=1123.932,149.823,-60.588,-179.536,8.708,149.556
C08657=1123.927,150.072,-60.610,-179.533,8.712,149.556
C08658=1123.923,150.321,-60.632,-179.531,8.715,149.556
C08659=1123.918,150.570,-60.654,-179.528,8.720,149.556
C08660=1123.914,150.819,-60.676,-179.525,8.723,149.556
C08661=1123.908,151.068,-60.697,-179.523,8.727,149.556
C08662=1123.904,151.317,-60.719,-179.521,8.730,149.557
C08663=1123.899,151.566,-60.741,-179.518,8.734,149.557
C08664=1123.894,151.815,-60.762,-179.515,8.738,149.557
C08665=1123.890,152.064,-60.784,-179.513,8.741,149.557
C08666=1123.885,152.313,-60.806,-179.511,8.744,149.557
C08667=1123.881,152.562,-60.828,-179.508,8.749,149.557
C08668=1123.876,152.811,-60.850,-179.506,8.752,149.558
C08669=1123.871,153.060,-60.871,-179.504,8.755,149.558
C08670=1123.867,153.309,-60.893,-179.500,8.759,149.558
C08671=1123.862,153.558,-60.915,-179.498,8.763,149.558
C08672=1123.857,153.807,-60.938,-179.496,8.766,149.558
C08673=1123.852,154.056,-60.959,-179.493,8.770,149.558
C08674=1123.848,154.305,-60.982,-179.491,8.773,149.559
C08675=1123.843,154.554,-61.003,-179.488,8.777,149.559
C08676=1123.839,154.803,-61.025,-179.486,8.780,149.559
C08677=1123.834,155.052,-61.047,-179.483,8.784,149.559
C08678=1123.830,155.301,-61.070,-179.481,8.787,149.559
C08679=1123.824,155.550,-61.092,-179.479,8.791,149.559
C08680=1123.820,155.799,-61.114,-179.477,8.794,149.559
C08681=1123.815,156.048,-61.136,-179.473,8.798,149.559
C08682=1123.811,156.297,-61.158,-179.471,8.801,149.560
C08683=1123.807,156.546,-61.180,-179.469,8.804,149.560
C08684=1123.801,156.795,-61.203,-179.467,8.808,149.560
C08685=1123.797,157.044,-61.225,-179.464,8.811,149.560
C08686=1123.793,157.258,-61.244,-179.462,8.814,149.560
C08687=1123.789,157.472,-61.263,-179.460,8.817,149.560
C08688=1123.785,157.686,-61.282,-179.458,8.820,149.560
C08689=1123.781,157.901,-61.301,-179.455,8.823,149.560
C08690=1123.777,158.115,-61.320,-179.454,8.826,149.560
C08691=1123.773,158.329,-61.339,-179.451,8.829,149.560
C08692=1123.769,158.543,-61.358,-179.450,8.832,149.561
C08693=1123.764,158.757,-61.378,-179.447,8.835,149.561
C08694=1123.760,159.007,-61.400,-179.445,8.838,149.561
C08695=1123.756,159.255,-61.422,-179.443,8.841,149.561
C08696=1123.751,159.504,-61.445,-179.440,8.844,149.561
C08697=1123.746,159.754,-61.467,-179.438,8.848,149.561
C08698=1123.742,160.002,-61.489,-179.435,8.851,149.561
C08699=1123.737,160.251,-61.512,-179.433,8.854,149.561
C08700=1123.733,160.500,-61.534,-179.431,8.858,149.562
C08701=1123.728,160.749,-61.556,-179.428,8.862,149.562
C08702=1123.723,160.998,-61.579,-179.425,8.865,149.562
C08703=1123.719,161.247,-61.602,-179.423,8.868,149.562
C08704=1123.714,161.496,-61.623,-179.421,8.871,149.562
C08705=1123.709,161.745,-61.647,-179.418,8.874,149.562
C08706=1123.705,161.994,-61.669,-179.416,8.878,149.562
C08707=1123.700,162.243,-61.692,-179.413,8.881,149.562
C08708=1123.696,162.492,-61.714,-179.411,8.884,149.562
C08709=1123.692,162.741,-61.736,-179.409,8.888,149.562
C08710=1123.686,162.990,-61.759,-179.406,8.891,149.563
C08711=1123.682,163.238,-61.782,-179.404,8.894,149.563
C08712=1123.677,163.488,-61.804,-179.402,8.897,149.563
C08713=1123.673,163.737,-61.827,-179.399,8.900,149.563
C08714=1123.668,163.986,-61.849,-179.397,8.903,149.563
C08715=1123.664,164.234,-61.872,-179.395,8.907,149.563
C08716=1123.659,164.483,-61.895,-179.392,8.910,149.563
C08717=1123.654,164.732,-61.917,-179.390,8.912,149.563
C08718=1123.649,164.981,-61.940,-179.388,8.916,149.563
C08719=1123.645,165.230,-61.963,-179.386,8.919,149.563
C08720=1123.640,165.479,-61.986,-179.383,8.922,149.563
C08721=1123.636,165.727,-62.008,-179.381,8.926,149.564
C08722=1123.631,165.976,-62.032,-179.378,8.929,149.564
C08723=1123.627,166.226,-62.054,-179.376,8.932,149.564
C08724=1123.622,166.475,-62.077,-179.373,8.935,149.564
C08725=1123.618,166.723,-62.099,-179.371,8.938,149.564
C08726=1123.613,166.972,-62.122,-179.369,8.941,149.564
C08727=1123.608,167.222,-62.145,-179.366,8.945,149.564
C08728=1123.604,167.470,-62.168,-179.365,8.947,149.564
C08729=1123.599,167.719,-62.191,-179.362,8.950,149.564
C08730=1123.594,167.968,-62.213,-179.360,8.954,149.564
C08731=1123.590,168.217,-62.237,-179.357,8.957,149.564
C08732=1123.585,168.466,-62.260,-179.355,8.960,149.565
C08733=1123.581,168.715,-62.283,-179.353,8.963,149.565
C08734=1123.576,168.964,-62.306,-179.351,8.966,149.565
C08735=1123.571,169.213,-62.328,-179.348,8.969,149.565
C08736=1123.567,169.461,-62.351,-179.346,8.972,149.565
C08737=1123.562,169.710,-62.374,-179.344,8.975,149.565
C08738=1123.557,169.959,-62.398,-179.341,8.978,149.565
C08739=1123.553,170.208,-62.421,-179.340,8.981,149.565
C08740=1123.548,170.457,-62.444,-179.337,8.984,149.565
C08741=1123.543,170.706,-62.467,-179.335,8.987,149.565
C08742=1123.540,170.920,-62.486,-179.333,8.990,149.565
C08743=1123.536,171.134,-62.506,-179.331,8.993,149.566
C08744=1123.532,171.348,-62.527,-179.329,8.995,149.566
C08745=1123.528,171.563,-62.546,-179.327,8.998,149.566
C08746=1123.524,171.776,-62.566,-179.325,9.000,149.566
C08747=1123.520,171.990,-62.586,-179.323,9.003,149.566
C08748=1123.516,172.205,-62.606,-179.321,9.006,149.566
C08749=1123.512,172.419,-62.626,-179.319,9.008,149.566
C08750=1123.508,172.668,-62.649,-179.316,9.011,149.566
C08751=1123.503,172.917,-62.672,-179.315,9.014,149.566
C08752=1123.498,173.166,-62.696,-179.312,9.017,149.566
C08753=1123.493,173.414,-62.718,-179.310,9.020,149.566
C08754=1123.489,173.663,-62.741,-179.308,9.024,149.567
C08755=1123.484,173.912,-62.765,-179.306,9.026,149.567
C08756=1123.480,174.161,-62.788,-179.303,9.029,149.567
C08757=1123.475,174.410,-62.811,-179.301,9.032,149.567
C08758=1123.470,174.659,-62.835,-179.299,9.035,149.567
C08759=1123.466,174.908,-62.857,-179.297,9.038,149.567
C08760=1123.462,175.156,-62.882,-179.294,9.041,149.567
C08761=1123.457,175.405,-62.905,-179.293,9.044,149.567
C08762=1123.453,175.654,-62.928,-179.290,9.047,149.567
C08763=1123.448,175.903,-62.952,-179.288,9.050,149.567
C08764=1123.443,176.152,-62.975,-179.286,9.053,149.568
C08765=1123.438,176.401,-62.998,-179.284,9.056,149.568
C08766=1123.434,176.650,-63.021,-179.281,9.059,149.568
C08767=1123.430,176.898,-63.045,-179.280,9.062,149.568
C08768=1123.425,177.147,-63.069,-179.277,9.065,149.568
C08769=1123.421,177.396,-63.092,-179.275,9.068,149.568
C08770=1123.416,177.645,-63.115,-179.273,9.071,149.568
C08771=1123.412,177.894,-63.139,-179.271,9.074,149.568
C08772=1123.407,178.143,-63.163,-179.269,9.076,149.568
C08773=1123.402,178.392,-63.186,-179.267,9.080,149.569
C08774=1123.397,178.641,-63.209,-179.264,9.083,149.569
C08775=1123.393,178.889,-63.233,-179.262,9.085,149.569
C08776=1123.388,179.138,-63.257,-179.260,9.089,149.569
C08777=1123.384,179.387,-63.280,-179.258,9.092,149.569
C08778=1123.379,179.636,-63.304,-179.255,9.095,149.569
C08779=1123.375,179.885,-63.328,-179.252,9.098,149.569
C08780=1123.370,180.134,-63.351,-179.249,9.101,149.569
C08781=1123.366,180.382,-63.375,-179.247,9.104,149.569
C08782=1123.361,180.631,-63.398,-179.244,9.108,149.569
C08783=1123.356,180.880,-63.422,-179.241,9.111,149.569
C08784=1123.352,181.129,-63.446,-179.238,9.114,149.569
C08785=1123.347,181.378,-63.469,-179.235,9.118,149.569
C08786=1123.343,181.626,-63.493,-179.232,9.121,149.569
C08787=1123.338,181.875,-63.517,-179.230,9.124,149.569
C08788=1123.334,182.124,-63.541,-179.227,9.127,149.569
C08789=1123.329,182.373,-63.564,-179.224,9.130,149.569
C08790=1123.325,182.622,-63.589,-179.221,9.134,149.569
C08791=1123.320,182.871,-63.612,-179.219,9.137,149.569
C08792=1123.316,183.119,-63.636,-179.216,9.140,149.569
C08793=1123.311,183.368,-63.659,-179.214,9.143,149.569
C08794=1123.307,183.617,-63.683,-179.211,9.146,149.569
C08795=1123.302,183.866,-63.707,-179.208,9.149,149.569
C08796=1123.297,184.115,-63.731,-179.206,9.152,149.569
C08797=1123.293,184.364,-63.756,-179.203,9.155,149.569
C08798=1123.289,184.577,-63.776,-179.201,9.158,149.569
C08799=1123.286,184.792,-63.796,-179.199,9.161,149.569
C08800=1123.281,185.006,-63.817,-179.196,9.163,149.569
C08801=1123.277,185.220,-63.838,-179.195,9.165,149.569
C08802=1123.274,185.433,-63.858,-179.192,9.168,149.569
C08803=1123.270,185.648,-63.879,-179.190,9.171,149.569
C08804=1123.266,185.861,-63.900,-179.188,9.173,149.569
C08805=1123.262,186.076,-63.921,-179.186,9.175,149.569
C08806=1123.257,186.324,-63.945,-179.184,9.178,149.569
C08807=1123.253,186.573,-63.968,-179.181,9.181,149.569
C08808=1123.248,186.821,-63.992,-179.179,9.185,149.569
C08809=1123.244,187.071,-64.017,-179.176,9.187,149.569
C08810=1123.239,187.320,-64.041,-179.174,9.190,149.569
C08811=1123.234,187.568,-64.065,-179.171,9.193,149.569
C08812=1123.230,187.817,-64.089,-179.169,9.196,149.569
C08813=1123.225,188.065,-64.113,-179.167,9.198,149.569
C08814=1123.221,188.315,-64.138,-179.164,9.201,149.569
C08815=1123.216,188.564,-64.161,-179.163,9.204,149.569
C08816=1123.212,188.812,-64.185,-179.160,9.207,149.569
C08817=1123.207,189.061,-64.210,-179.157,9.210,149.569
C08818=1123.203,189.310,-64.234,-179.156,9.212,149.569
C08819=1123.199,189.558,-64.259,-179.153,9.215,149.569
C08820=1123.193,189.808,-64.282,-179.151,9.218,149.569
C08821=1123.189,190.056,-64.307,-179.149,9.221,149.570
C08822=1123.185,190.305,-64.331,-179.147,9.223,149.570
C08823=1123.180,190.554,-64.356,-179.145,9.227,149.570
C08824=1123.176,190.802,-64.380,-179.143,9.229,149.570
C08825=1123.170,191.051,-64.404,-179.141,9.231,149.570
C08826=1123.167,191.300,-64.429,-179.138,9.234,149.570
C08827=1123.162,191.549,-64.453,-179.136,9.237,149.570
C08828=1123.157,191.797,-64.478,-179.134,9.240,149.570
C08829=1123.153,192.046,-64.502,-179.132,9.242,149.570
C08830=1123.149,192.295,-64.526,-179.131,9.245,149.570
C08831=1123.144,192.543,-64.551,-179.129,9.247,149.570
C08832=1123.139,192.792,-64.575,-179.127,9.251,149.571
C08833=1123.135,193.041,-64.600,-179.125,9.253,149.571
C08834=1123.131,193.290,-64.624,-179.123,9.255,149.571
C08835=1123.125,193.538,-64.649,-179.121,9.259,149.571
C08836=1123.122,193.788,-64.673,-179.119,9.261,149.571
C08837=1123.116,194.036,-64.698,-179.117,9.263,149.571
C08838=1123.112,194.285,-64.722,-179.115,9.266,149.571
C08839=1123.108,194.534,-64.746,-179.114,9.268,149.571
C08840=1123.103,194.783,-64.771,-179.112,9.271,149.571
C08841=1123.099,195.031,-64.795,-179.110,9.274,149.572
C08842=1123.094,195.280,-64.820,-179.108,9.277,149.572
C08843=1123.090,195.529,-64.844,-179.106,9.279,149.572
C08844=1123.085,195.778,-64.869,-179.105,9.282,149.572
C08845=1123.081,196.027,-64.893,-179.103,9.284,149.572
C08846=1123.076,196.275,-64.919,-179.101,9.287,149.572
C08847=1123.072,196.524,-64.943,-179.098,9.291,149.572
C08848=1123.067,196.773,-64.968,-179.095,9.294,149.572
C08849=1123.063,197.021,-64.992,-179.091,9.298,149.572
C08850=1123.058,197.270,-65.017,-179.087,9.301,149.572
C08851=1123.053,197.519,-65.041,-179.084,9.305,149.572
C08852=1123.050,197.768,-65.067,-179.081,9.309,149.572
C08853=1123.044,198.016,-65.091,-179.078,9.312,149.572
C08854=1123.041,198.230,-65.113,-179.074,9.315,149.572
C08855=1123.037,198.444,-65.134,-179.072,9.318,149.572
C08856=1123.033,198.658,-65.155,-179.069,9.321,149.571
C08857=1123.029,198.872,-65.176,-179.066,9.324,149.571
C08858=1123.026,199.086,-65.198,-179.063,9.327,149.571
C08859=1123.021,199.299,-65.219,-179.060,9.329,149.571
C08860=1123.018,199.513,-65.240,-179.057,9.332,149.571
C08861=1123.014,199.727,-65.262,-179.054,9.335,149.571
C08862=1123.009,199.976,-65.286,-179.051,9.339,149.571
C08863=1123.005,200.225,-65.312,-179.048,9.342,149.571
C08864=1123.000,200.473,-65.336,-179.045,9.345,149.571
C08865=1122.996,200.723,-65.361,-179.042,9.348,149.571
C08866=1122.991,200.971,-65.387,-179.038,9.351,149.570
C08867=1122.987,201.220,-65.411,-179.035,9.354,149.570
C08868=1122.982,201.468,-65.436,-179.032,9.358,149.570
C08869=1122.978,201.717,-65.461,-179.029,9.361,149.570
C08870=1122.973,201.965,-65.487,-179.025,9.364,149.570
C08871=1122.969,202.215,-65.511,-179.023,9.367,149.570
C08872=1122.964,202.463,-65.537,-179.020,9.370,149.570
C08873=1122.960,202.712,-65.562,-179.016,9.373,149.570
C08874=1122.956,202.961,-65.587,-179.013,9.376,149.569
C08875=1122.951,203.209,-65.612,-179.010,9.379,149.569
C08876=1122.947,203.458,-65.637,-179.008,9.382,149.569
C08877=1122.942,203.706,-65.663,-179.004,9.385,149.569
C08878=1122.938,203.956,-65.688,-179.001,9.388,149.569
C08879=1122.933,204.204,-65.713,-178.998,9.391,149.569
C08880=1122.928,204.453,-65.738,-178.995,9.394,149.569
C08881=1122.924,204.701,-65.763,-178.993,9.397,149.569
C08882=1122.920,204.950,-65.789,-178.990,9.399,149.569
C08883=1122.915,205.199,-65.814,-178.987,9.402,149.569
C08884=1122.911,205.447,-65.839,-178.984,9.405,149.568
C08885=1122.906,205.696,-65.865,-178.981,9.408,149.568
C08886=1122.902,205.944,-65.890,-178.978,9.411,149.568
C08887=1122.897,206.194,-65.915,-178.975,9.413,149.568
C08888=1122.893,206.442,-65.941,-178.973,9.417,149.568
C08889=1122.888,206.691,-65.966,-178.970,9.419,149.568
C08890=1122.885,206.939,-65.992,-178.967,9.422,149.568
C08891=1122.880,207.188,-66.017,-178.964,9.425,149.568
C08892=1122.875,207.437,-66.042,-178.961,9.428,149.568
C08893=1122.871,207.685,-66.068,-178.959,9.431,149.568
C08894=1122.866,207.933,-66.093,-178.957,9.433,149.568
C08895=1122.862,208.182,-66.119,-178.954,9.436,149.568
C08896=1122.857,208.432,-66.144,-178.951,9.439,149.568
C08897=1122.853,208.680,-66.169,-178.949,9.442,149.568
C08898=1122.848,208.929,-66.195,-178.946,9.445,149.568
C08899=1122.844,209.177,-66.221,-178.944,9.447,149.568
C08900=1122.839,209.426,-66.246,-178.941,9.450,149.568
C08901=1122.835,209.674,-66.272,-178.938,9.453,149.568
C08902=1122.831,209.923,-66.298,-178.936,9.455,149.568
C08903=1122.827,210.172,-66.323,-178.934,9.458,149.568
C08904=1122.822,210.420,-66.349,-178.931,9.461,149.568
C08905=1122.818,210.669,-66.375,-178.929,9.464,149.568
C08906=1122.813,210.918,-66.400,-178.927,9.467,149.568
C08907=1122.808,211.166,-66.426,-178.925,9.469,149.568
C08908=1122.804,211.415,-66.452,-178.922,9.472,149.568
C08909=1122.799,211.664,-66.478,-178.920,9.474,149.568
C08910=1122.796,211.878,-66.499,-178.918,9.477,149.568
C08911=1122.792,212.091,-66.522,-178.916,9.479,149.568
C08912=1122.788,212.305,-66.544,-178.915,9.482,149.568
C08913=1122.784,212.519,-66.566,-178.913,9.484,149.568
C08914=1122.780,212.733,-66.588,-178.911,9.486,149.568
C08915=1122.776,212.946,-66.611,-178.909,9.489,149.568
C08916=1122.773,213.160,-66.632,-178.907,9.491,149.568
C08917=1122.769,213.374,-66.655,-178.906,9.494,149.569
C08918=1122.764,213.622,-66.680,-178.903,9.497,149.569
C08919=1122.760,213.871,-66.706,-178.901,9.499,149.569
C08920=1122.755,214.120,-66.732,-178.900,9.502,149.569
C08921=1122.751,214.369,-66.757,-178.897,9.505,149.569
C08922=1122.747,214.617,-66.784,-178.896,9.508,149.569
C08923=1122.742,214.865,-66.810,-178.893,9.511,149.569
C08924=1122.737,215.114,-66.836,-178.892,9.513,149.569
C08925=1122.733,215.363,-66.861,-178.889,9.517,149.570
C08926=1122.729,215.612,-66.887,-178.888,9.519,149.570
C08927=1122.725,215.860,-66.913,-178.885,9.522,149.570
C08928=1122.720,216.108,-66.940,-178.884,9.525,149.570
C08929=1122.715,216.357,-66.965,-178.881,9.528,149.570
C08930=1122.711,216.606,-66.991,-178.879,9.530,149.570
C08931=1122.707,216.855,-67.017,-178.877,9.534,149.570
C08932=1122.703,217.103,-67.043,-178.874,9.537,149.570
C08933=1122.698,217.352,-67.070,-178.873,9.539,149.570
C08934=1122.693,217.600,-67.095,-178.870,9.543,149.571
C08935=1122.689,217.849,-67.121,-178.868,9.546,149.571
C08936=1122.685,218.097,-67.147,-178.865,9.549,149.571
C08937=1122.680,218.346,-67.174,-178.864,9.551,149.571
C08938=1122.676,218.595,-67.199,-178.861,9.555,149.571
C08939=1122.672,218.843,-67.226,-178.859,9.558,149.571
C08940=1122.667,219.092,-67.252,-178.856,9.561,149.571
C08941=1122.662,219.340,-67.278,-178.854,9.564,149.571
C08942=1122.658,219.589,-67.304,-178.851,9.567,149.571
C08943=1122.654,219.837,-67.330,-178.849,9.570,149.572
C08944=1122.649,220.086,-67.357,-178.847,9.573,149.572
C08945=1122.645,220.335,-67.383,-178.845,9.576,149.572
C08946=1122.641,220.583,-67.408,-178.842,9.579,149.572
C08947=1122.636,220.832,-67.435,-178.840,9.582,149.572
C08948=1122.632,221.081,-67.461,-178.837,9.585,149.572
C08949=1122.627,221.329,-67.488,-178.835,9.588,149.572
C08950=1122.623,221.578,-67.514,-178.832,9.592,149.572
C08951=1122.619,221.826,-67.540,-178.829,9.595,149.572
C08952=1122.614,222.075,-67.566,-178.826,9.598,149.572
C08953=1122.610,222.323,-67.593,-178.824,9.602,149.572
C08954=1122.605,222.572,-67.619,-178.821,9.605,149.572
C08955=1122.601,222.820,-67.646,-178.819,9.608,149.572
C08956=1122.596,223.069,-67.672,-178.816,9.611,149.572
C08957=1122.592,223.317,-67.699,-178.813,9.614,149.572
C08958=1122.588,223.566,-67.724,-178.810,9.617,149.572
C08959=1122.583,223.815,-67.751,-178.808,9.621,149.572
C08960=1122.579,224.063,-67.778,-178.805,9.624,149.573
C08961=1122.574,224.312,-67.804,-178.802,9.628,149.573
C08962=1122.570,224.560,-67.831,-178.799,9.630,149.572
C08963=1122.566,224.809,-67.858,-178.797,9.633,149.573
C08964=1122.561,225.058,-67.883,-178.793,9.637,149.573
C08965=1122.557,225.306,-67.911,-178.790,9.640,149.572
C08966=1122.553,225.520,-67.933,-178.788,9.643,149.573
C08967=1122.549,225.733,-67.956,-178.785,9.646,149.573
C08968=1122.546,225.947,-67.979,-178.783,9.648,149.572
C08969=1122.542,226.160,-68.002,-178.781,9.651,149.573
C08970=1122.538,226.374,-68.025,-178.778,9.654,149.572
C08971=1122.534,226.588,-68.048,-178.775,9.657,149.572
C08972=1122.530,226.801,-68.071,-178.772,9.660,149.572
C08973=1122.527,227.016,-68.094,-178.770,9.662,149.572
C08974=1122.523,227.264,-68.120,-178.767,9.666,149.572
C08975=1122.518,227.512,-68.147,-178.764,9.669,149.572
C08976=1122.513,227.761,-68.174,-178.761,9.672,149.572
C08977=1122.510,228.009,-68.201,-178.757,9.676,149.572
C08978=1122.505,228.258,-68.227,-178.754,9.679,149.572
C08979=1122.500,228.507,-68.254,-178.751,9.683,149.572
C08980=1122.496,228.755,-68.281,-178.748,9.685,149.572
C08981=1122.491,229.003,-68.308,-178.744,9.689,149.572
C08982=1122.487,229.252,-68.335,-178.741,9.692,149.572
C08983=1122.483,229.500,-68.361,-178.738,9.695,149.572
C08984=1122.479,229.749,-68.389,-178.734,9.699,149.571
C08985=1122.474,229.998,-68.416,-178.731,9.702,149.571
C08986=1122.470,230.246,-68.442,-178.728,9.705,149.571
C08987=1122.465,230.494,-68.469,-178.724,9.708,149.571
C08988=1122.461,230.743,-68.496,-178.721,9.712,149.571
C08989=1122.456,230.991,-68.523,-178.718,9.715,149.571
C08990=1122.452,231.240,-68.550,-178.714,9.718,149.571
C08991=1122.448,231.489,-68.577,-178.711,9.721,149.571
C08992=1122.444,231.737,-68.604,-178.708,9.724,149.571
C08993=1122.439,231.986,-68.631,-178.705,9.727,149.570
C08994=1122.434,232.234,-68.658,-178.702,9.730,149.570
C08995=1122.431,232.482,-68.686,-178.699,9.733,149.570
C08996=1122.426,232.730,-68.713,-178.695,9.736,149.570
C08997=1122.422,232.979,-68.740,-178.692,9.739,149.570
C08998=1122.417,233.228,-68.767,-178.689,9.742,149.570
C08999=1122.413,233.476,-68.794,-178.686,9.745,149.570
C09000=1122.408,233.725,-68.821,-178.683,9.747,149.570
C09001=1122.404,233.973,-68.848,-178.680,9.751,149.569
C09002=1122.400,234.222,-68.876,-178.677,9.754,149.569
C09003=1122.396,234.470,-68.903,-178.674,9.756,149.569
C09004=1122.391,234.719,-68.930,-178.671,9.759,149.569
C09005=1122.387,234.967,-68.958,-178.668,9.762,149.569
C09006=1122.383,235.216,-68.985,-178.665,9.765,149.569
C09007=1122.378,235.464,-69.012,-178.662,9.768,149.569
C09008=1122.374,235.712,-69.040,-178.659,9.770,149.569
C09009=1122.369,235.961,-69.067,-178.657,9.772,149.569
C09010=1122.365,236.210,-69.095,-178.654,9.775,149.568
C09011=1122.360,236.458,-69.122,-178.651,9.778,149.568
C09012=1122.356,236.706,-69.149,-178.648,9.781,149.568
C09013=1122.352,236.955,-69.177,-178.645,9.783,149.568
C09014=1122.347,237.203,-69.205,-178.644,9.786,149.568
C09015=1122.343,237.452,-69.232,-178.641,9.788,149.568
C09016=1122.338,237.700,-69.259,-178.638,9.791,149.568
C09017=1122.334,237.949,-69.287,-178.635,9.794,149.568
C09018=1122.330,238.197,-69.314,-178.632,9.796,149.568
C09019=1122.325,238.445,-69.342,-178.630,9.799,149.568
C09020=1122.321,238.694,-69.369,-178.628,9.801,149.568
C09021=1122.317,238.942,-69.397,-178.625,9.804,149.567
C09022=1122.314,239.156,-69.421,-178.623,9.806,149.568
C09023=1122.310,239.370,-69.444,-178.620,9.808,149.567
C09024=1122.305,239.583,-69.468,-178.618,9.810,149.567
C09025=1122.302,239.797,-69.492,-178.616,9.812,149.567
C09026=1122.298,240.010,-69.515,-178.614,9.815,149.567
C09027=1122.295,240.224,-69.539,-178.612,9.817,149.567
C09028=1122.291,240.437,-69.563,-178.610,9.819,149.567
C09029=1122.288,240.651,-69.587,-178.608,9.821,149.567
C09030=1122.283,240.899,-69.614,-178.606,9.823,149.567
C09031=1122.279,241.147,-69.642,-178.604,9.825,149.567
C09032=1122.275,241.396,-69.669,-178.601,9.828,149.567
C09033=1122.270,241.644,-69.697,-178.599,9.830,149.567
C09034=1122.265,241.892,-69.725,-178.597,9.833,149.567
C09035=1122.261,242.141,-69.753,-178.594,9.836,149.567
C09036=1122.257,242.389,-69.780,-178.592,9.838,149.567
C09037=1122.253,242.638,-69.809,-178.590,9.840,149.567
C09038=1122.248,242.886,-69.836,-178.588,9.842,149.567
C09039=1122.244,243.134,-69.863,-178.586,9.844,149.567
C09040=1122.240,243.383,-69.892,-178.583,9.848,149.567
C09041=1122.235,243.632,-69.919,-178.581,9.850,149.567
C09042=1122.231,243.880,-69.947,-178.580,9.852,149.567
C09043=1122.227,244.128,-69.975,-178.578,9.855,149.567
C09044=1122.223,244.377,-70.003,-178.576,9.857,149.567
C09045=1122.218,244.625,-70.030,-178.574,9.859,149.567
C09046=1122.213,244.873,-70.059,-178.572,9.862,149.567
C09047=1122.210,245.122,-70.087,-178.570,9.864,149.567
C09048=1122.205,245.370,-70.114,-178.568,9.866,149.567
C09049=1122.201,245.619,-70.142,-178.566,9.869,149.568
C09050=1122.196,245.867,-70.170,-178.564,9.871,149.568
C09051=1122.192,246.116,-70.199,-178.562,9.873,149.568
C09052=1122.188,246.364,-70.226,-178.561,9.876,149.568
C09053=1122.184,246.613,-70.254,-178.560,9.877,149.568
C09054=1122.179,246.861,-70.282,-178.558,9.880,149.568
C09055=1122.174,247.109,-70.310,-178.556,9.882,149.568
C09056=1122.171,247.357,-70.338,-178.554,9.885,149.568
C09057=1122.166,247.605,-70.366,-178.551,9.888,149.568
C09058=1122.162,247.854,-70.395,-178.545,9.893,149.568
C09059=1122.157,248.103,-70.422,-178.539,9.898,149.568
C09060=1122.153,248.351,-70.450,-178.534,9.903,149.567
C09061=1122.148,248.599,-70.478,-178.529,9.906,149.567
C09062=1122.145,248.848,-70.506,-178.523,9.911,149.566
C09063=1122.140,249.096,-70.534,-178.518,9.914,149.566
C09064=1122.136,249.345,-70.563,-178.514,9.918,149.566
C09065=1122.132,249.593,-70.591,-178.509,9.922,149.565
C09066=1122.127,249.842,-70.619,-178.504,9.926,149.565
C09067=1122.123,250.090,-70.648,-178.500,9.929,149.565
C09068=1122.119,250.337,-70.676,-178.496,9.932,149.564
C09069=1122.115,250.586,-70.705,-178.492,9.935,149.564
C09070=1122.110,250.834,-70.733,-178.488,9.939,149.564
C09071=1122.106,251.083,-70.761,-178.484,9.942,149.564
C09072=1122.102,251.332,-70.789,-178.481,9.945,149.563
C09073=1122.097,251.580,-70.818,-178.477,9.948,149.563
C09074=1122.094,251.828,-70.847,-178.474,9.950,149.563
C09075=1122.089,252.077,-70.875,-178.471,9.953,149.563
C09076=1122.085,252.325,-70.903,-178.469,9.955,149.562
C09077=1122.080,252.573,-70.932,-178.466,9.958,149.562
C09078=1122.077,252.786,-70.956,-178.463,9.960,149.562
C09079=1122.073,253.000,-70.981,-178.461,9.962,149.562
C09080=1122.069,253.213,-71.006,-178.460,9.963,149.562
C09081=1122.066,253.426,-71.029,-178.457,9.965,149.562
C09082=1122.062,253.640,-71.054,-178.456,9.967,149.562
C09083=1122.058,253.854,-71.079,-178.454,9.968,149.562
C09084=1122.054,254.066,-71.104,-178.453,9.969,149.562
C09085=1122.051,254.280,-71.128,-178.452,9.971,149.562
C09086=1122.047,254.528,-71.157,-178.450,9.973,149.562
C09087=1122.042,254.776,-71.185,-178.449,9.975,149.562
C09088=1122.038,255.025,-71.214,-178.448,9.976,149.562
C09089=1122.034,255.274,-71.243,-178.447,9.978,149.562
C09090=1122.029,255.521,-71.271,-178.447,9.979,149.563
C09091=1122.025,255.770,-71.300,-178.446,9.981,149.563
C09092=1122.021,256.018,-71.328,-178.446,9.982,149.563
C09093=1122.016,256.266,-71.357,-178.443,9.984,149.563
C09094=1122.012,256.515,-71.385,-178.440,9.987,149.563
C09095=1122.008,256.763,-71.414,-178.437,9.990,149.563
C09096=1122.004,257.012,-71.443,-178.434,9.993,149.563
C09097=1121.999,257.260,-71.472,-178.432,9.996,149.563
C09098=1121.995,257.508,-71.500,-178.429,9.999,149.563
C09099=1121.991,257.757,-71.529,-178.426,10.001,149.562
C09100=1121.987,258.004,-71.558,-178.423,10.004,149.562
C09101=1121.982,258.253,-71.586,-178.420,10.007,149.562
C09102=1121.978,258.502,-71.616,-178.416,10.010,149.562
C09103=1121.974,258.750,-71.644,-178.413,10.013,149.562
C09104=1121.970,258.998,-71.673,-178.410,10.016,149.562
C09105=1121.965,259.247,-71.702,-178.408,10.019,149.562
C09106=1121.961,259.495,-71.731,-178.405,10.021,149.562
C09107=1121.957,259.743,-71.759,-178.402,10.024,149.562
C09108=1121.952,259.991,-71.788,-178.398,10.028,149.562
C09109=1121.948,260.239,-71.818,-178.395,10.030,149.561
C09110=1121.944,260.488,-71.847,-178.392,10.033,149.561
C09111=1121.940,260.736,-71.875,-178.389,10.037,149.561
C09112=1121.935,260.984,-71.904,-178.385,10.039,149.561
C09113=1121.931,261.233,-71.933,-178.382,10.042,149.561
C09114=1121.927,261.481,-71.963,-178.379,10.045,149.561
C09115=1121.922,261.730,-71.991,-178.376,10.048,149.561
C09116=1121.919,261.978,-72.020,-178.372,10.051,149.560
C09117=1121.914,262.225,-72.049,-178.369,10.054,149.560
C09118=1121.910,262.474,-72.079,-178.366,10.057,149.560
C09119=1121.905,262.722,-72.108,-178.363,10.059,149.560
C09120=1121.901,262.971,-72.137,-178.359,10.063,149.560
C09121=1121.897,263.219,-72.167,-178.356,10.065,149.559
C09122=1121.893,263.467,-72.196,-178.352,10.069,149.559
